   // sequencer 1
   INITIAL_STEP "No mode active":   // S1, max time T#10S, warning time T#7S
              N    #mode.activeMode:="mode_0_not_selected"
   END_STEP
   TRANSITION Trans1 FROM "No mode active" TO "Return to base position active"   // T1
      := #mode.button.basic.request.visibility AND #mode.button.basic.request.button;
   END_TRANSITION
   TRANSITION Trans6 FROM "No mode active" TO "Manual mode active"   // T6
      := NOT #mode.switch.auto AND "DB_Eks_Instance".Status.Global.AnyValidKey AND #iSafetyOKmanual;
   END_TRANSITION
   STEP "Return to base position active":   // S2, max time T#10S, warning time T#7S
              N    #mode.activeMode:="mode_2_base"
   END_STEP
   TRANSITION Trans2 FROM "Return to base position active" TO "Base position reached"   // T2
      := #iBasePosition;
   END_TRANSITION
   TRANSITION Trans5 FROM "Return to base position active" TO Done   // T5
      := NOT #iSafetyOKauto OR ((NOT #iBaseInManualMode OR #mode.switch.poloautomaActivated) AND NOT #mode.switch.auto) OR (#iBaseInManualMode AND #mode.switch.auto AND NOT #mode.switch.poloautomaActivated) OR #F_TRIG_semiauto_switch.Q;
   END_TRANSITION
   STEP "Base position reached":   // S3, max time T#10S, warning time T#7S
              N    #mode.activeMode:="mode_2_base"
   END_STEP
   TRANSITION Trans3 FROM "Base position reached" TO "Automatic mode active"   // T3
      := (#mode.button.auto.startRequest.visibility AND #mode.button.auto.startRequest.button) OR #mode.switch.poloautomaActivated;
   END_TRANSITION
   TRANSITION Trans8 FROM "Base position reached" TO Done   // T8
      := NOT #iSafetyOKauto OR (NOT #iBaseInManualMode AND NOT #mode.switch.auto) OR NOT #iBasePosition OR #F_TRIG_switchAuto.Q;
   END_TRANSITION
   STEP "Automatic mode active":   // S4, max time T#10S, warning time T#7S
              N    #mode.activeMode:="mode_3_automat"
   END_STEP
   TRANSITION Trans4 FROM "Automatic mode active" TO Done   // T4
      := NOT "AlwaysTRUE";
   END_TRANSITION
   TRANSITION Trans9 FROM "Automatic mode active" TO Done   // T9
      := NOT #iSafetyOKauto OR NOT #mode.switch.auto;
   END_TRANSITION
   TRANSITION Trans12 FROM "Automatic mode active" TO "R1 EXT off during auto"   // T12
      := NOT "iR1ext";
   END_TRANSITION
   STEP "Manual mode active":   // S5, max time T#10S, warning time T#7S
              N    #mode.activeMode:="mode_1_manual"
   END_STEP
   TRANSITION Trans7 FROM "Manual mode active" TO Done   // T7
      := #mode.switch.auto OR NOT "DB_Eks_Instance".Status.Global.AnyValidKey OR NOT #iSafetyOKmanual;
   END_TRANSITION
   TRANSITION Trans10 FROM "Manual mode active" TO "Return to base position active"   // T10, jump
      := #mode.button.basic.request.visibility AND #mode.button.basic.request.button;
   END_TRANSITION
   STEP Done:   // S6, max time T#10S, warning time T#7S
   END_STEP
   TRANSITION Trans11 FROM Done TO "No mode active"   // T11, jump
      := TRUE;
   END_TRANSITION
   STEP "R1 EXT off during auto":   // S7, max time T#10S, warning time T#7S
   END_STEP
   TRANSITION Trans13 FROM "R1 EXT off during auto" TO Done   // T13
      := TRUE;
   END_TRANSITION

   // permanent post-instructions
   NETWORK 1
   TITLE = semiauto mode
      IF ((#mode.activeMode = "mode_2_base") OR (#mode.activeMode = "mode_3_automat")) AND #mode.switch.poloautomaActivated THEN
          #mode.activeMode := "mode_4_semiautomat";
      END_IF;
   NETWORK 2
   TITLE = previous mode
      #mode.modeChanged := #mode.activeMode <> #PrevMode;
      #PrevMode := #mode.activeMode;
END_FUNCTION_BLOCK

FUNCTION_BLOCK "Lamps"   // FB7, LAD
{ S7_Optimized_Access := 'TRUE' }
VERSION : 0.1
// stored: AutoNumber true, IsIECCheckEnabled false, IsRetainMemResEnabled false, MemoryReserve 100, SetENOAutomatically false, UDAEnableTagReadback false
   VAR
      R_TRIG_Instance { S7_SetPoint := 'True'} : R_TRIG;
      IEC_Timer_0_Instance { S7_SetPoint := 'True'} : TON_TIME;
   END_VAR
BEGIN

REGION Network 1: Lighthouse lamps
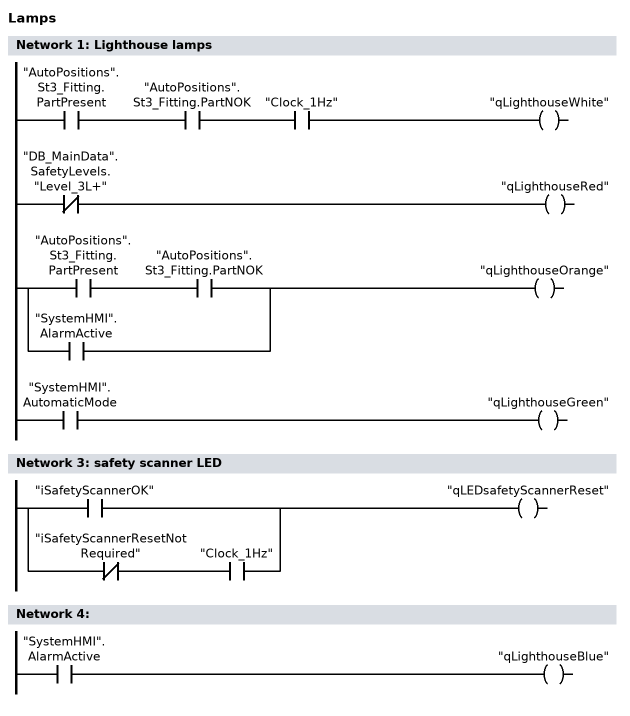
   RUNG wire#powerrail
      Contact( "AutoPositions".St3_Fitting.PartPresent )
      Contact( "AutoPositions".St3_Fitting.PartNOK )
      Contact( "Clock_1Hz" )
      Coil( "qLighthouseWhite" )
   END_RUNG
   RUNG wire#powerrail
      I_Contact( "DB_MainData".SafetyLevels."Level_3L+" )
      Coil( "qLighthouseRed" )
   END_RUNG
   RUNG wire#powerrail
      Contact( "AutoPositions".St3_Fitting.PartPresent )
      Contact( "AutoPositions".St3_Fitting.PartNOK )
      wire#w1
      Coil( "qLighthouseOrange" )
   END_RUNG
   RUNG wire#powerrail
      Contact( "SystemHMI".AlarmActive )
   END_RUNG wire#w1
   RUNG wire#powerrail
      Contact( "SystemHMI".AutomaticMode )
      Coil( "qLighthouseGreen" )
   END_RUNG
   // the same network as SCL:
   "qLighthouseWhite" := "AutoPositions".St3_Fitting.PartPresent AND "AutoPositions".St3_Fitting.PartNOK AND "Clock_1Hz";
   "qLighthouseRed" := NOT "DB_MainData".SafetyLevels."Level_3L+";
   "qLighthouseOrange" := ("AutoPositions".St3_Fitting.PartPresent AND "AutoPositions".St3_Fitting.PartNOK) OR "SystemHMI".AlarmActive;
   "qLighthouseGreen" := "SystemHMI".AutomaticMode;
END_REGION

REGION Network 2 (SCL): Alarm LED on OP
   //red button hmi
   "qResetAlarm" := "SystemHMI".AlarmActiveBlinking  AND "Clock_1Hz";
END_REGION

REGION Network 3: safety scanner LED
   RUNG wire#powerrail
      Contact( "iSafetyScannerOK" )
      wire#w1
      Coil( "qLEDsafetyScannerReset" )
   END_RUNG
   RUNG wire#powerrail
      I_Contact( "iSafetyScannerResetNotRequired" )
      Contact( "Clock_1Hz" )
   END_RUNG wire#w1
   // the same network as SCL:
   "qLEDsafetyScannerReset" := "iSafetyScannerOK" OR (NOT "iSafetyScannerResetNotRequired" AND "Clock_1Hz");
END_REGION

REGION Network 4
   RUNG wire#powerrail
      Contact( "SystemHMI".AlarmActive )
      Coil( "qLighthouseBlue" )
   END_RUNG
   // the same network as SCL:
   "qLighthouseBlue" := "SystemHMI".AlarmActive;
END_REGION
END_FUNCTION_BLOCK

FUNCTION "FC_READING_MAIN" : Void   // FC304, LAD
{ S7_Optimized_Access := 'TRUE' }
VERSION : 0.1
// stored: AutoNumber false, IsIECCheckEnabled false, SetENOAutomatically false, UDAEnableTagReadback false
BEGIN

REGION Network 1: Dataman readers block calls
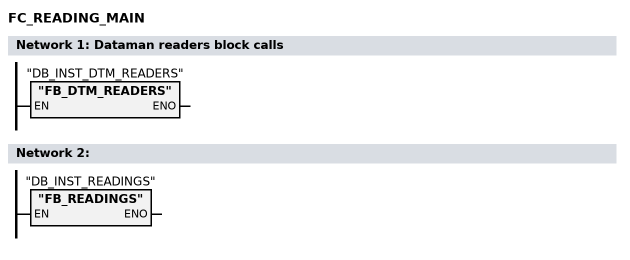
   RUNG wire#powerrail
      "DB_INST_DTM_READERS"()
   END_RUNG
   // the same network as SCL:
   "DB_INST_DTM_READERS"();   // "FB_DTM_READERS"
END_REGION

REGION Network 2
   RUNG wire#powerrail
      "DB_INST_READINGS"()
   END_RUNG
   // the same network as SCL:
   "DB_INST_READINGS"();   // "FB_READINGS"
END_REGION
END_FUNCTION

FUNCTION_BLOCK "FB_DTM_READERS"
{ S7_Optimized_Access := 'TRUE' }
VERSION : 0.1
   VAR 
      READER { S7_SetPoint := 'False'} : Array[1..5] of "FB_DTM";
   END_VAR


BEGIN
	//Call block reader 1
	#READER[1](TriggerReady:= "DM_SMLH-TriggerReady",
	           TriggerAck:="DM_SMLH-TriggerAck",
	           ResultsAvailable:="DM_SMLH-Results Available",
	           ResultID:="DM_SMLH-ResultID",
	           ResultCode:="DM_SMLH-Result Code",
	           ResultLenght:="DM_SMLH-Result Length",
	           ResultData:="DM_SMLH-ResultData",
	           TriggerEnable=>"DM_SMLH-TriggerEnable",
	           Trigger=>"DM_SMLH-Trigger",
	           ResultsAck=>"DM_SMLH-ResultsAck"
	          );
	
	//Call block reader 2
	          #READER[2](TriggerReady := "DM_SMRH-TriggerReady",
	           TriggerAck := "DM_SMRH-TriggerAck",
	           ResultsAvailable := "DM_SMRH-Results Available",
	           ResultID := "DM_SMRH-ResultID",
	           ResultCode := "DM_SMRH-Result Code",
	           ResultLenght := "DM_SMRH-Result Length",
	           ResultData := "DM_SMRH-ResultData",
	           TriggerEnable => "DM_SMRH-TriggerEnable",
	           Trigger => "DM_SMRH-Trigger",
	           ResultsAck => "DM_SMRH-ResultsAck"
	           );
	
	//Call block reader 3
	           #READER[3](TriggerReady:= "DM_FT-TriggerReady",
	           TriggerAck := "DM_FT-TriggerAck",
	           ResultsAvailable := "DM_FT-Results Available",
	           ResultID := "DM_FT-ResultID",
	           ResultCode := "DM_FT-Result Code",
	           ResultLenght := "DM_FT-Result Length",
	           ResultData := "DM_FT-ResultData",
	           TriggerEnable => "DM_FT-TriggerEnable",
	           Trigger => "DM_FT-Trigger",
	           ResultsAck => "DM_FT-ResultsAck");
	
	//Call block reader 4
	#READER[4](TriggerReady:= "DM_RT-TriggerReady",
	           TriggerAck := "DM_RT-TriggerAck",
	           ResultsAvailable := "DM_RT-Results Available",
	           ResultID := "DM_RT-ResultID",
	           ResultCode := "DM_RT-Result Code",
	           ResultLenght := "DM_RT-Result Length",
	           ResultData := "DM_RT-ResultData",
	           TriggerEnable => "DM_RT-TriggerEnable",
	           Trigger => "DM_RT-Trigger",
	           ResultsAck => "DM_RT-ResultsAck");
	
	
END_FUNCTION_BLOCK

FUNCTION_BLOCK "FB_DTM"   // FB301, LAD
{ S7_Optimized_Access := 'TRUE' }
VERSION : 0.1
// stored: AutoNumber false, IsIECCheckEnabled false, IsRetainMemResEnabled false, MemoryReserve 100, SetENOAutomatically false, UDAEnableTagReadback false
   VAR_INPUT
      Req : Bool;
      TriggerReady : Bool;
      TriggerAck : Bool;
      ResultsAvailable : Bool;
      ResultID : Word;
      ResultCode : Word;
      ResultLenght : Word;
      ResultData : "udt_DTM_resultData";
   END_VAR
   VAR_OUTPUT
      TriggerEnable : Bool;
      Trigger : Bool;
      ResultsAck : Bool;
      DataStr : String;
   END_VAR
   VAR
      ResultPending { ExternalAccessible := 'False'; ExternalVisible := 'False'; ExternalWritable := 'False'} : Bool;
      LatestResults { ExternalAccessible := 'False'; ExternalVisible := 'False'; ExternalWritable := 'False'} : Struct
         ID { ExternalAccessible := 'False'; ExternalVisible := 'False'; ExternalWritable := 'False'} : Int;
         Flags { ExternalAccessible := 'False'; ExternalVisible := 'False'; ExternalWritable := 'False'} : Int;
         Length { ExternalAccessible := 'False'; ExternalVisible := 'False'; ExternalWritable := 'False'} : Int;
         Value { ExternalAccessible := 'False'; ExternalVisible := 'False'; ExternalWritable := 'False'} : Array[0..63] of Byte;
      END_STRUCT;
   END_VAR
   VAR CONSTANT
      test : Bool := true;
   END_VAR
   VAR_TEMP   // added for the SCL form of the ladder/FBD networks
      _w1 : Bool;
   END_VAR
BEGIN

REGION Network 1: DataMan Acquisition Control Module
   // Make sure triggering is enabled
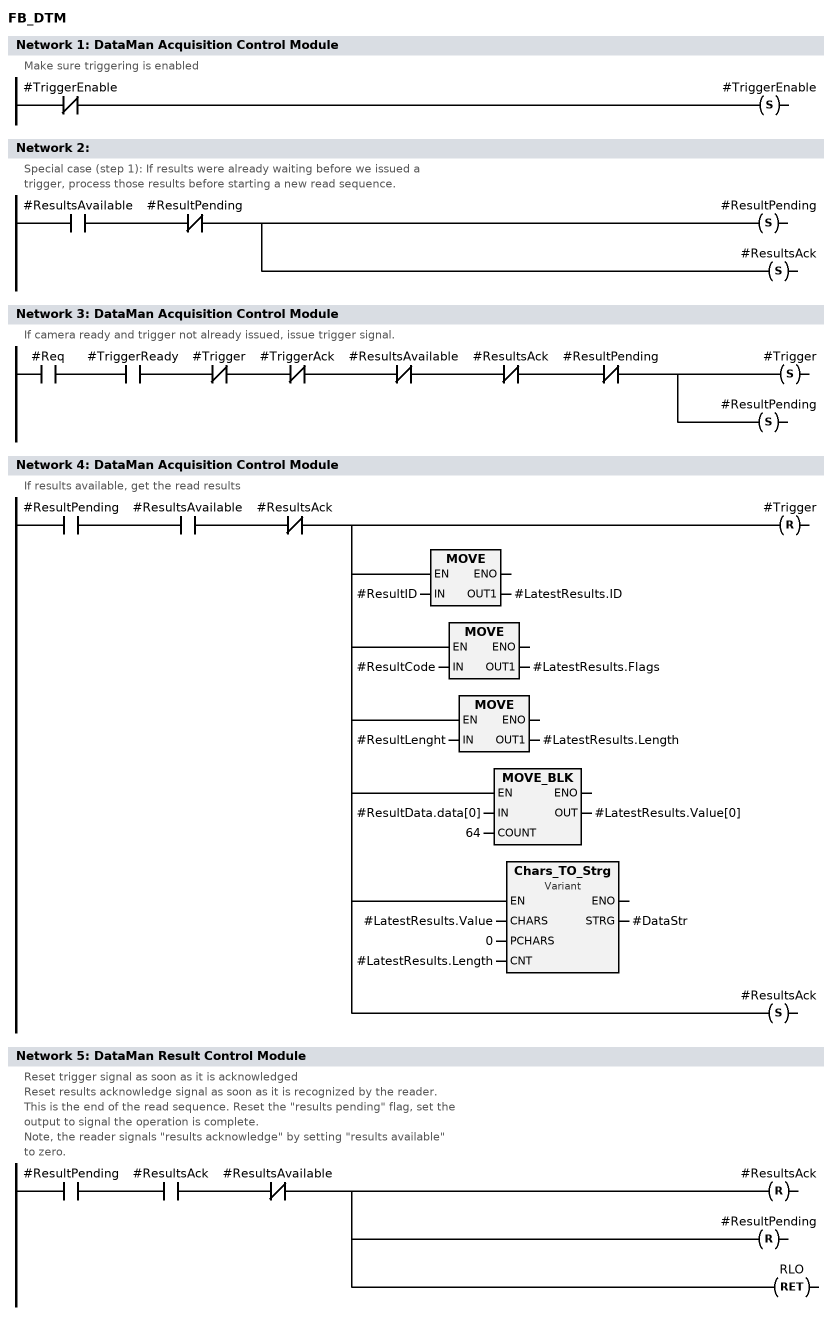
   RUNG wire#powerrail
      I_Contact( #TriggerEnable )
      S_Coil( #TriggerEnable )
   END_RUNG
   // the same network as SCL:
   IF NOT #TriggerEnable THEN #TriggerEnable := TRUE; END_IF;
END_REGION

REGION Network 2
   // Special case (step 1): If results were already waiting before we issued a 
   // trigger, process those results before starting a new read sequence.
   RUNG wire#powerrail
      Contact( #ResultsAvailable )
      I_Contact( #ResultPending )
      wire#w1
      S_Coil( #ResultPending )
   END_RUNG
   RUNG wire#w1
      S_Coil( #ResultsAck )
   END_RUNG
   // the same network as SCL:
   #_w1 := #ResultsAvailable AND NOT #ResultPending;
   IF #_w1 THEN
       #ResultPending := TRUE;
       #ResultsAck := TRUE;
   END_IF;
END_REGION

REGION Network 3: DataMan Acquisition Control Module
   // If camera ready and trigger not already issued, issue trigger signal.
   RUNG wire#powerrail
      Contact( #Req )
      Contact( #TriggerReady )
      I_Contact( #Trigger )
      I_Contact( #TriggerAck )
      I_Contact( #ResultsAvailable )
      I_Contact( #ResultsAck )
      I_Contact( #ResultPending )
      wire#w1
      S_Coil( #Trigger )
   END_RUNG
   RUNG wire#w1
      S_Coil( #ResultPending )
   END_RUNG
   // the same network as SCL:
   #_w1 := #Req AND #TriggerReady AND NOT #Trigger AND NOT #TriggerAck AND NOT #ResultsAvailable AND NOT #ResultsAck AND NOT #ResultPending;
   IF #_w1 THEN
       #Trigger := TRUE;
       #ResultPending := TRUE;
   END_IF;
END_REGION

REGION Network 4: DataMan Acquisition Control Module
   // If results available, get the read results
   IF #ResultPending AND #ResultsAvailable AND NOT #ResultsAck THEN
       #Trigger := FALSE;
       #LatestResults.ID := #ResultID;
       #LatestResults.Flags := #ResultCode;
       #LatestResults.Length := #ResultLenght;
       MOVE_BLK(IN := #ResultData.data[0], COUNT := 64, OUT => #LatestResults.Value[0]);
       Chars_TO_Strg(Chars := #LatestResults.Value, pChars := 0, Cnt := #LatestResults.Length, Strg => #DataStr);
       #ResultsAck := TRUE;
   END_IF;
END_REGION

REGION Network 5: DataMan Result Control Module
   // Reset trigger signal as soon as it is acknowledged 
   // Reset results acknowledge signal as soon as it is recognized by the reader.
   // 
   // This is the end of the read sequence. Reset the "results pending" flag, set the 
   // output to signal the operation is complete.
   // 
   // Note, the reader signals "results acknowledge" by setting "results available" 
   // to zero.
   #_w1 := #ResultPending AND #ResultsAck AND NOT #ResultsAvailable;
   IF #_w1 THEN
       #ResultsAck := FALSE;
       #ResultPending := FALSE;
       ENO := TRUE;
       RETURN;
   END_IF;
END_REGION
END_FUNCTION_BLOCK

FUNCTION_BLOCK "FB_READINGS"
{ S7_Optimized_Access := 'FALSE' }
VERSION : 0.1
   VAR 
      Reading : Array[1.."MaxDataReading"] of Struct
         Done : Bool;
         OK : Bool;
         NOK : Bool;
         Scan : String[70];
         NFP : String[30];
         IJC : Array[1.."NumberOfmessages"] of Struct
            SendMsg : Bool;
            Done : Bool;
            Answer : Int;
            State : USInt;
         END_STRUCT;
      END_STRUCT;
      ReadingsDone : Bool;
      Errors : Array[1..2] of Word;
      Error { ExternalAccessible := 'False'; ExternalVisible := 'False'; ExternalWritable := 'False'} AT Errors : Array[1..2, 1..16] of Bool;
   END_VAR

   VAR_TEMP 
      lctr1 : Int;
      lctr2 : Int;
      tempHolder : String;
      blankStr : String;
      NumberOfReadings : Int;
      eType : Int;   // Error type 1:reading, 2:IJCore
      count : Int;
   END_VAR

   VAR CONSTANT 
      NotUsed : USInt := 0;
      MasterNFP : USInt := 2;
      SecondaryNFP : USInt := 3;
      Component : USInt := 4;
   END_VAR


BEGIN
	//TITLE = 'READINGS'
	//AUTHOR: RAUL ROBINS
	//CREATED ON: 03/24/2023
	//VERSION: 1.0
	
	#NumberOfReadings := "DB_ProductionProgramActual".Program.NumberOfReadings;
	
	REGION Read code
	    
	    //Read request
	    IF "DevicesData".scanner.start THEN
	        FOR #lctr1 := 1 TO #NumberOfReadings DO
	            IF "DB_ProductionProgramActual".Program.Readings[#lctr1].Enable AND
	                NOT #Reading[#lctr1].Done THEN
	                "DB_INST_DTM_READERS".READER["DB_ProductionProgramActual".Program.Readings[#lctr1].ReaderNumber].Req := TRUE;
	            END_IF;
	            IF "DB_INST_DTM_READERS".READER["DB_ProductionProgramActual".Program.Readings[#lctr1].ReaderNumber].ResultsAvailable AND
	                "DB_INST_DTM_READERS".READER["DB_ProductionProgramActual".Program.Readings[#lctr1].ReaderNumber].ResultLenght <> 0 THEN
	                "DB_INST_DTM_READERS".READER["DB_ProductionProgramActual".Program.Readings[#lctr1].ReaderNumber].Req := FALSE;
	                #Reading[#lctr1].Done := TRUE;
	            END_IF;
	            
	            //Results
	            IF #Reading[#lctr1].Done THEN
	                //Compare strings
	                #tempHolder := MID(IN := "DB_INST_DTM_READERS".READER["DB_ProductionProgramActual".Program.Readings[#lctr1].ReaderNumber].DataStr,
	                                   L := LEN("DB_ProductionProgramActual".Program.Readings[#lctr1].ReferenceToFound),
	                                   P := "DB_ProductionProgramActual".Program.Readings[#lctr1].ReferenceStartPosition);
	                
	                IF #tempHolder = "DB_ProductionProgramActual".Program.Readings[#lctr1].ReferenceToFound THEN
	                    //Results OK
	                    #Reading[#lctr1].Scan := "DB_INST_DTM_READERS".READER["DB_ProductionProgramActual".Program.Readings[#lctr1].ReaderNumber].DataStr;
	                    #Reading[#lctr1].OK := TRUE;
	                    #Reading[#lctr1].NOK := FALSE;
	                    
	                    
	                    //Copy  NFP 
	                    //Master NFP
	                    IF "DB_ProductionProgramActual".Program.Readings[#lctr1].LabelType = 2 THEN
	                        #Reading[#lctr1].NFP := LEFT(IN := "DB_INST_DTM_READERS".READER["DB_ProductionProgramActual".Program.Readings[#lctr1].ReaderNumber].DataStr, L := 30);
	                        //Secondary NFP
	                    ELSIF "DB_ProductionProgramActual".Program.Readings[#lctr1].LabelType = 3 THEN
	                        //Linked to created NFP
	                        IF "DB_ProductionProgramActual".Program.Readings[1].MasterReadingNumber > 0 THEN
	                            ;
	                            //Linked to readed NFP
	                        ELSIF "DB_ProductionProgramActual".Program.Readings[1].LinkedMasterNumber > 0 THEN
	                            #Reading[#lctr1].NFP := #Reading["DB_ProductionProgramActual".Program.Readings[#lctr1].LinkedMasterNumber].NFP;
	                        END_IF;
	                        
	                    END_IF;
	                ELSE
	                    //Results NOK
	                    #Reading[#lctr1].OK := FALSE;
	                    #Reading[#lctr1].NOK := TRUE;
	                    #Reading[#lctr1].Scan := #blankStr;
	                END_IF;
	            END_IF;
	            //Count readings ok
	            IF #Reading[#lctr1].OK AND (#Reading[#lctr1].Scan <> #blankStr) OR NOT "DB_ProductionProgramActual".Program.Readings[#lctr1].Enable THEN
	                #count += 1;
	            END_IF;
	            IF #count = "DB_ProductionProgramActual".Program.NumberOfReadings THEN
	                #ReadingsDone := TRUE;
	            END_IF;
	            //Copy readings to buffer data
	            IF "sq_carousel_insertion_st1"."Set part present".X THEN
	                "AutoPositions".St1_Table1.Readings[#lctr1].Scan := #Reading[#lctr1].Scan;
	            END_IF;
	            
	            
	        END_FOR;
	    END_IF;
	    
	    
	    
	END_REGION
	
	REGION IJCore
	    FOR #lctr1 := 1 TO #NumberOfReadings DO
	        //TRACE
	        FOR #lctr2 := 1 TO 5 DO
	            CASE "DB_ProductionProgramActual".Program.Readings[#lctr1].Message[#lctr2].MessageType OF
	                "STA":
	                    "FC_READING_IJC_STA"(Req := #Reading[#lctr1].OK,
	                                         MessageNumber := "DB_ProductionProgramActual".Program.Readings[#lctr1].Message[#lctr2].MessageFlagNumber,
	                                         TraceabilityMode := "DB_MAIN_IJCORE".Mode,
	                                         NFP := #Reading[#lctr1].Scan,
	                                         ErrReset := "AlwaysTRUE",
	                                         MessageDone => #Reading[#lctr1].IJC[#lctr2].Done,
	                                         Answer := #Reading[#lctr1].IJC[#lctr2].Answer,
	                                         State := #Reading[#lctr1].IJC[#lctr2].State);
	                    
	                "PFC":
	                    "FC_TRACE_PFC"(Req := "DB_MAIN_IJCORE".CMD.PFC,
	                                   MessageNumber := "DB_ProductionProgramActual".Program.Readings[#lctr1].Message[#lctr2].MessageFlagNumber,
	                                   TraceabilityMode := "DB_MAIN_IJCORE".Mode,
	                                   NFP := "AutoPositions".St3_Fitting.Readings["DB_ProductionProgramActual".Program.Readings[#lctr1].MasterReadingNumber].Scan,
	                                   Kanban := "DB_ProductionProgramActual".Program.FaureciaNumber,
	                                   ErrReset := TRUE,
	                                   MessageDone => #Reading[#lctr1].IJC[#lctr2].Done,
	                                   Answer => #Reading[#lctr1].IJC[#lctr2].Answer,
	                                   State := #Reading[#lctr1].IJC[#lctr2].State);
	                    
	                "TRR":
	                    "FC_TRACE_TRR"(Req := "DB_MAIN_IJCORE".CMD.TRR,
	                                   MessageNumber := "DB_ProductionProgramActual".Program.Readings[#lctr1].Message[#lctr2].MessageFlagNumber,
	                                   TraceabilityMode := "DB_MAIN_IJCORE".Mode,
	                                   NFP := "AutoPositions".St3_Fitting.Readings["DB_ProductionProgramActual".Program.Readings[#lctr1].MasterReadingNumber].Scan,
	                                   ProcessStatus := 1,
	                                   NumberOfProcess := 1,
	                                   ErrReset := TRUE,
	                                   MessageDone => #Reading[#lctr1].IJC[#lctr2].Done,
	                                   Answer => #Reading[#lctr1].IJC[#lctr2].Answer,
	                                   State := #Reading[#lctr1].IJC[#lctr2].State);
	                    
	                "TRC":
	                    IF "DB_ProductionProgramActual".Program.Readings[#lctr1].MasterReadingNumber > 0 THEN
	                        "FC_READING_IJC_TRC"(Req := "DB_MAIN_IJCORE".CMD.TRC,
	                                             MessageNumber := "DB_ProductionProgramActual".Program.Readings[#lctr1].Message[#lctr2].MessageFlagNumber,
	                                             TraceabilityMode := "DB_MAIN_IJCORE".Mode,
	                                             NFP := #Reading["DB_ProductionProgramActual".Program.Readings[#lctr1].MasterReadingNumber].Scan,
	                                             Scan := #Reading[#lctr1].Scan,
	                                             ErrReset := TRUE,
	                                             MessageDone => #Reading[#lctr1].IJC[#lctr2].Done,
	                                             Answer := #Reading[#lctr1].IJC[#lctr2].Answer,
	                                             State := #Reading[#lctr1].IJC[#lctr2].State);
	                    END_IF;
	                ELSE:
	                    ;
	                    
	            END_CASE;
	            
	        END_FOR;
	    END_FOR;
	    
	END_REGION
	
	
	
	
	REGION Clear Data
	    IF NOT "DevicesData".scanner.start THEN
	        FOR #lctr1 := 1 TO "MaxDataReading" DO
	            "DB_INST_DTM_READERS".READER["DB_ProductionProgramActual".Program.Readings[#lctr1].ReaderNumber].Req := FALSE;
	            #Reading[#lctr1].Done := FALSE;
	            #Reading[#lctr1].OK := FALSE;
	            #Reading[#lctr1].NOK := FALSE;
	            #ReadingsDone := FALSE;
	            #Reading[#lctr1].Scan := #blankStr;
	        END_FOR;
	    END_IF;
	END_REGION
	
	// REGION Error Management
	//     #eType := 1;
	//     FOR #lctr1 := 1 TO #NumberOfReadings DO
	//         IF #Reading[#lctr1].NOK THEN
	//             #Error[#eType, 1] := TRUE;
	//         END_IF;
	
	//         //IJCore Errors
	//         FOR #lctr2 := 1 TO "NumberOfIJCoreMessages" DO
	//             #eType := 2;
	//             CASE #Reading[#lctr1].IJC[#lctr2].Answer OF
	//                 -2:  // NFP not founded
	//                     #Error[#eType, 1] := TRUE;
	//                 -3:  //Part number NOT inside BOM
	//                     #Error[#eType, 2] := TRUE;
	//                 -4: // PFC not ok
	//                     #Error[#eType, 3] := TRUE;
	//                 -5: //Component already used
	//                     #Error[#eType, 4] := TRUE;
	//                 -6: //Module already used
	//                     #Error[#eType, 5] := true;
	//                 -10: //Status NOK from previous operation
	//                     #Error[#eType, 6] := true;
	//             END_CASE;
	//         END_FOR;
	//     END_FOR;
	
	//     FOR #lctr1 := 1 TO 2 DO
	//         #Errors[#lctr1] := SWAP(#Errors[#lctr1]);
	//     END_FOR;
	// END_REGION
	
	
	
	
	
	
END_FUNCTION_BLOCK

FUNCTION "FC_TRACE_TRR" : Void
{ S7_Optimized_Access := 'TRUE' }
VERSION : 0.1
   VAR_INPUT 
      Req : Bool;   // Request message
      MessageNumber : DInt;   // Message number
      TraceabilityMode : Int;   // Tracability mode
      NFP : String;
      ProcessStatus : USInt;
      NumberOfProcess : USInt;
      ErrReset : Bool;
   END_VAR

   VAR_OUTPUT 
      MessageDone : Bool;
      Answer : Int;
   END_VAR

   VAR_IN_OUT 
      State : USInt;
   END_VAR

   VAR_TEMP 
      SEND_OFFSET : Struct
         SW : DInt;
         MSG : DInt;
      END_STRUCT;
      REC_OFFSET : Struct
         SW : DInt;
         MSG : DInt;
         ANS : DInt;
      END_STRUCT;
      IDB : Int;
      i : Int;
      j : Int;
      k : Int;
      CNT : Int;
      CNT_STR : String[2];
      MSG : DInt;
      ErrCode : Int;
   END_VAR

   VAR CONSTANT 
      "DB" : Byte := 16#84;
      CLEAR : Word := 16#0000;
      MINUS1 : Word := 16#FFFF;
      PLUS1 : Word := 16#0001;
      DB_REC : DB_ANY := 1006;
      DB_SEND : DB_ANY := 1005;
      Blank : String := '';
   END_VAR


BEGIN
	//TITLE = 'IJCORE PROTOCOL'
	//AUTHOR: RAUL ROBINS
	//CREATED ON: 03/24/2023
	//VERSION: 3.0
	
	
	
	IF #MessageNumber < 1  THEN
	    RETURN;
	END_IF;
	
	
	
	
	IF NOT #Req THEN // Error Reset
	    #State := 0;
	END_IF;
	
	#SEND_OFFSET.SW := (#MessageNumber * 2) + 2; //Calc message send sw offset
	#SEND_OFFSET.MSG := ((#MessageNumber - 1) * 80) + 604; // Calc send message offset
	#REC_OFFSET.SW := (#MessageNumber - 1) * 2; // Calc receive sw offset
	#REC_OFFSET.ANS := ((#MessageNumber - 1) * 32) + 600; // Calc receive answer offset
	#REC_OFFSET.MSG := ((#MessageNumber - 1) * 32) + 602; // Calc receive message offset
	
	
	CASE #State OF
	    0: // Initial State
	        #MessageDone := FALSE;
	        #Answer := 0;
	
	        POKE(area := #DB, //Clear send flag
	             dbNumber := #DB_SEND,
	             byteOffset := #SEND_OFFSET.SW,
	             value := #MINUS1);
	        POKE(area := #DB, //Clear receive flag
	             dbNumber := #DB_REC,
	             byteOffset := #REC_OFFSET.SW,
	             value := #MINUS1);
	     
	        #State := 10; ///Transition to state 10
	        
	    10: // Wait for start command
	        IF #Req THEN //If start command active
	            
	            POKE(area := #DB, //Clear send flag
	                 dbNumber := #DB_SEND,
	                 byteOffset := #SEND_OFFSET.SW,
	                 value := #MINUS1);
	            POKE(area := #DB, //Clear receive flag
	                 dbNumber := #DB_REC,
	                 byteOffset := #REC_OFFSET.SW,
	                 value := #MINUS1);
	            POKE(area := #DB, // Clear answer 
	                 dbNumber := #DB_REC,
	                 byteOffset := #REC_OFFSET.ANS,
	                 value := #CLEAR);
	            
	            FOR #i := 0 TO 79 BY 1 DO //Clear all send array
	                POKE(area := #DB,
	                     dbNumber := #DB_SEND,
	                     byteOffset := (#SEND_OFFSET.MSG + #i),
	                     value := '$00');
	            END_FOR;
	            FOR #i := 0 TO 29 BY 1 DO //Clear all receive array
	                POKE(area := #DB,
	                     dbNumber := #DB_REC,
	                     byteOffset := (#REC_OFFSET.MSG + #i),
	                     value := '$00');
	            END_FOR;
	            #State := 20; //Transition to state 20
	        END_IF;
	        
	    20: // Create message to send
	        FOR #i := 0 TO 7 BY 1 DO //Copy NFP to DB to send
	            POKE(area := #DB,
	                 dbNumber := #DB_SEND,
	                 byteOffset := (#SEND_OFFSET.MSG + #i),
	                 value := #NFP[#i + 1]);
	        END_FOR;
	                
	  
	                
	                POKE(area := #DB, //Set the process status of the message
	                     dbNumber := #DB_SEND,
	                     byteOffset := (#SEND_OFFSET.MSG + 8),
	                     value := USINT_TO_CHAR(#ProcessStatus + 48));
	                
	          
	        #State := 30; // Transition to state 30
	        
	    30: //Set flag to "1" to inform that PLC is ready to send (DB5 Ó 1005)
	        POKE(area := #DB,//Set flag to "1" to inform that PLC is ready to send
	             dbNumber := #DB_SEND,
	             byteOffset := #SEND_OFFSET.SW,
	             value := #PLUS1);
	        #State := 40; // Transition to state 40
	        
	        
	    40: //Wait to IJCORE response with "-1"
	        IF (PEEK_WORD(area := #DB, dbNumber := #DB_SEND, byteOffset := #SEND_OFFSET.SW) = #MINUS1)
	        THEN
	            #State := 50; // Transition to state 50
	        END_IF;
	        
	    50: //Check if IJCORE have answer from DB Receive
	        IF (PEEK_WORD(area := #DB, dbNumber := #DB_REC, byteOffset := #REC_OFFSET.SW) = #PLUS1)
	        THEN
	            #Answer := WORD_TO_INT(PEEK_WORD(area := #DB, dbNumber := #DB_REC, byteOffset := #REC_OFFSET.ANS)); //Copy answer from IJCORE
	
	            #State := 60; // Transition to state 100
	        END_IF;
	        
	    60: //Change Flag to "-1"
	        POKE(area := #DB, //Set "-1" to IJCORE
	             dbNumber := #DB_REC,
	             byteOffset := #REC_OFFSET.SW,
	             value := #MINUS1);
	        #State := 100; // Transition to state 100
	        
	        
	    100: //Sequence done
	        CASE #TraceabilityMode OF
	            1:// Full traceability
	                IF #Answer = 1 THEN
	                    #MessageDone := TRUE;
	                ELSE
	                    #MessageDone := FALSE;
	                END_IF;
	            2:// Traceability only
	                #MessageDone := TRUE;
	        END_CASE;
	        
	        IF NOT #Req THEN
	            #State := 0; // Transition to state 0
	        END_IF;
	END_CASE;
	
	
	
	
	
	
	
END_FUNCTION

ORGANIZATION_BLOCK "Startup"   // OB124, LAD, Startup
TITLE = "Complete Restart"
{ S7_Optimized_Access := 'TRUE' }
VERSION : 0.1
// stored: AutoNumber true, IsIECCheckEnabled false, SetENOAutomatically false
   VAR_INPUT
      LostRetentive : Bool;   // True if retentive data are lost
      LostRTC : Bool;   // True if date and time are lost
   END_VAR
BEGIN

REGION Network 1: Braketest or mastering requred
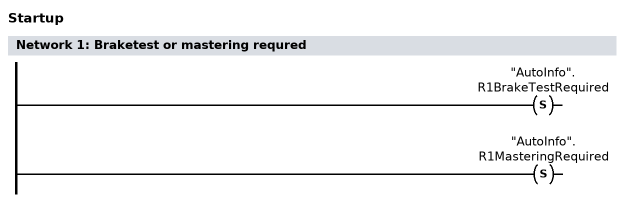
   RUNG wire#powerrail
      S_Coil( "AutoInfo".R1BrakeTestRequired )
   END_RUNG
   RUNG wire#powerrail
      S_Coil( "AutoInfo".R1MasteringRequired )
   END_RUNG
   // the same network as SCL:
   "AutoInfo".R1BrakeTestRequired := TRUE;
   "AutoInfo".R1MasteringRequired := TRUE;
END_REGION

REGION Network 2 (SCL)
       "DevicesData"."TA1-3MA".OverAcc := "StationParameters".Servo.OverAcc;
       "DevicesData"."TA1-3MA".OverDec := "StationParameters".Servo.OverDec;
       "DevicesData"."TA1-3MA".OverV := "StationParameters".Servo.OverV;
       "DevicesData"."TA1-3MA".Velocity := "StationParameters".Servo.Velocity;
END_REGION

REGION Network 3 (SCL)
   "setup_DB".minL := 100.0;
   "setup_DB".minR := "setup_DB".minL;
END_REGION
END_ORGANIZATION_BLOCK

ORGANIZATION_BLOCK "OB_IO_AccessError"   // OB122, LAD, IOAccessError
{ S7_Optimized_Access := 'TRUE' }
VERSION : 0.1
// stored: IsIECCheckEnabled false, SetENOAutomatically false
   VAR_INPUT
      BlockNr : UInt;   // Number of causing block
      Reaction : USInt;   // 0:ignore, 1:substitute, 2:skip
      Fault_ID : Byte;   // 16#42:reading, 16#43:writing
      BlockType : USInt;   // 16#01:OB, 16#02:FC, 16#03:FB, 16#04:SFC, 16#05:SFB, 16#06:DB: Type of block causing the error
      Area : USInt;   // 16#81:I, 16#82:Q: IO area where the IOaccess error occured
      DBNr : DB_ANY;   // Reserved for system
      Csg_OBNr : OB_ANY;   // Number of OB causing the error
      Csg_Prio : USInt;   // Priority of OB causing the error
      Width : USInt;   // 0:bit, 1:byte, 2:word, 3:dword, 4:lword
   END_VAR
BEGIN
END_ORGANIZATION_BLOCK

ORGANIZATION_BLOCK "OB_ProgrammingError"   // OB121, LAD, ProgrammingError
{ S7_Optimized_Access := 'TRUE' }
VERSION : 0.1
// stored: IsIECCheckEnabled false, SetENOAutomatically false
   VAR_INPUT
      BlockNr : UInt;   // Number of causing block
      Reaction : USInt;   // 0:ignore, 1:substitute, 2:skip
      Fault_ID : Byte;   // Fault identifier
      BlockType : USInt;   // 16#01:OB, 16#02:FC, 16#03:FB, 16#04:SFC, 16#05:SFB, 16#06:DB: Type of block causing the error
      Area : USInt;   // Area where the error occured
      DBNr : DB_ANY;   // DB number if Area = DB or DI
      Csg_OBNr : OB_ANY;   // Number of OB causing the error
      Csg_Prio : USInt;   // Priority of OB causing the error
      Width : USInt;   // 0:bit, 1:byte, 2:word, 3:dword, 4:lword
   END_VAR
BEGIN
END_ORGANIZATION_BLOCK

ORGANIZATION_BLOCK "OB_RackStationFailure"   // OB86, LAD, RackOrStationFailure
{ S7_Optimized_Access := 'TRUE' }
VERSION : 0.1
// stored: IsIECCheckEnabled false, SetENOAutomatically false
   VAR_INPUT
      LADDR : HW_DEVICE;   // Hardware identifier
      Event_Class : Byte;   // Event class
      Fault_ID : Byte;   // Fault identifier
   END_VAR
BEGIN
END_ORGANIZATION_BLOCK

ORGANIZATION_BLOCK "OB_Startup"   // OB100, LAD, Startup
TITLE = "Complete Restart"
{ S7_Optimized_Access := 'TRUE' }
VERSION : 0.1
// stored: AutoNumber true, IsIECCheckEnabled false, SetENOAutomatically false
   VAR_INPUT
      LostRetentive : Bool;   // True if retentive data are lost
      LostRTC : Bool;   // True if date and time are lost
   END_VAR
BEGIN
END_ORGANIZATION_BLOCK

ORGANIZATION_BLOCK "Diagnostic error interrupt"   // OB82, LAD, DiagnosticErrorInterrupt
{ S7_Optimized_Access := 'TRUE' }
VERSION : 0.1
// stored: IsIECCheckEnabled false, SetENOAutomatically false
   VAR_INPUT
      IO_State : Word;   // IO state of the HW object
      LADDR : HW_ANY;   // Hardware identifier
      Channel : UInt;   // Channel number
      MultiError : Bool;   // =true if more than one error is present
   END_VAR
BEGIN
END_ORGANIZATION_BLOCK

FUNCTION_BLOCK "CylinderINC"   // FB30, LAD
{ S7_Optimized_Access := 'FALSE' }
AUTHOR : Bodorik
FAMILY : RIV
NAME : Cylinder
VERSION : 0.9
// stored: AutoNumber false, IsIECCheckEnabled false, SetENOAutomatically false, UDAEnableTagReadback false
   VAR_INPUT
      POWER_OK : Bool;
      MOVE_BASIC : Bool;
      MOVE_WORK : Bool;
      MOVE_FREE : Bool;
      BASIC_POSITION : Bool;
      WORK_POSITION : Bool;
      TRIGGER : Bool;
      RESET : Bool;
      DELAY_BASIC : Time := T#1S;
      DELAY_WORK : Time := T#1S;
      DELAY_FREE : Time := T#1S;
      ERROR_TIME : Time := T#1S;
      ValveDelay : Time;
   END_VAR
   VAR_OUTPUT
      VALVE_BASIC : Bool;
      VALVE_WORK : Bool;
      CylinderStatus : "CylinderStatus";
      ERROR_BASIC : Bool;
      ERROR_WORK : Bool;
   END_VAR
   VAR_IN_OUT
      CylinderOperation : "CylinderOperation";
   END_VAR
   VAR DB_SPECIFIC
      "4l+Started" : Bool;
      InitCommandBP : Bool;
      InitCommandWP : Bool;
      BasicWorkStartWP : Bool;
      BasicWorkStartBP : Bool;
      work_valve : Bool;
      basic_valve : Bool;
      free_valve : Bool;
      baspos_error { S7_SetPoint := 'True'} : TON_TIME;
      workpos_error { S7_SetPoint := 'True'} : TON_TIME;
      baspos_delay { S7_SetPoint := 'True'} : TON_TIME;
      workpos_delay { S7_SetPoint := 'True'} : TON_TIME;
      CylinderOperationOld { S7_SetPoint := 'True'} : "CylinderOperation";
      IEC_Timer_0_Instance { S7_SetPoint := 'True'} : TP_TIME;
   END_VAR
   VAR
      R_TRIG_Instance { S7_SetPoint := 'True'} : R_TRIG;
   END_VAR
   VAR DB_SPECIFIC
      IEC_Timer_0_Instance_1 { S7_SetPoint := 'True'} : TP_TIME;
      IEC_Timer_0_Instance_2 { S7_SetPoint := 'True'} : TP_TIME;
      IEC_Timer_0_Instance_3 { S7_SetPoint := 'True'} : TON_TIME;
      IEC_Timer_0_Instance_4 { S7_SetPoint := 'True'} : TON_TIME;
   END_VAR
   VAR_TEMP
      et : Bool;
   END_VAR
   VAR_TEMP   // added for the SCL form of the ladder/FBD networks
      _w1 : Bool;
   END_VAR
BEGIN

REGION Network 1 (SCL): check new cylinder command
   //check if basic position req movement changed
   IF #CylinderOperation.ToBp <> #CylinderOperationOld.ToBp THEN
       #CylinderOperation.ToFp := false;
       #CylinderOperation.ToWp := false;
   END_IF;
   //check if work position req movement changed
   IF #CylinderOperation.ToWp <> #CylinderOperationOld.ToWp THEN
       #CylinderOperation.ToFp := false;
       #CylinderOperation.ToBp := false;
   END_IF;
   //check if free position req movement changed
   IF #CylinderOperation.ToFp <> #CylinderOperationOld.ToFp THEN
       #CylinderOperation.ToBp := false;
       #CylinderOperation.ToWp := false;
   END_IF;
   //store actual cylinder status to old
   #CylinderOperationOld := #CylinderOperation;
END_REGION

REGION Network 2: Start movement to basic position
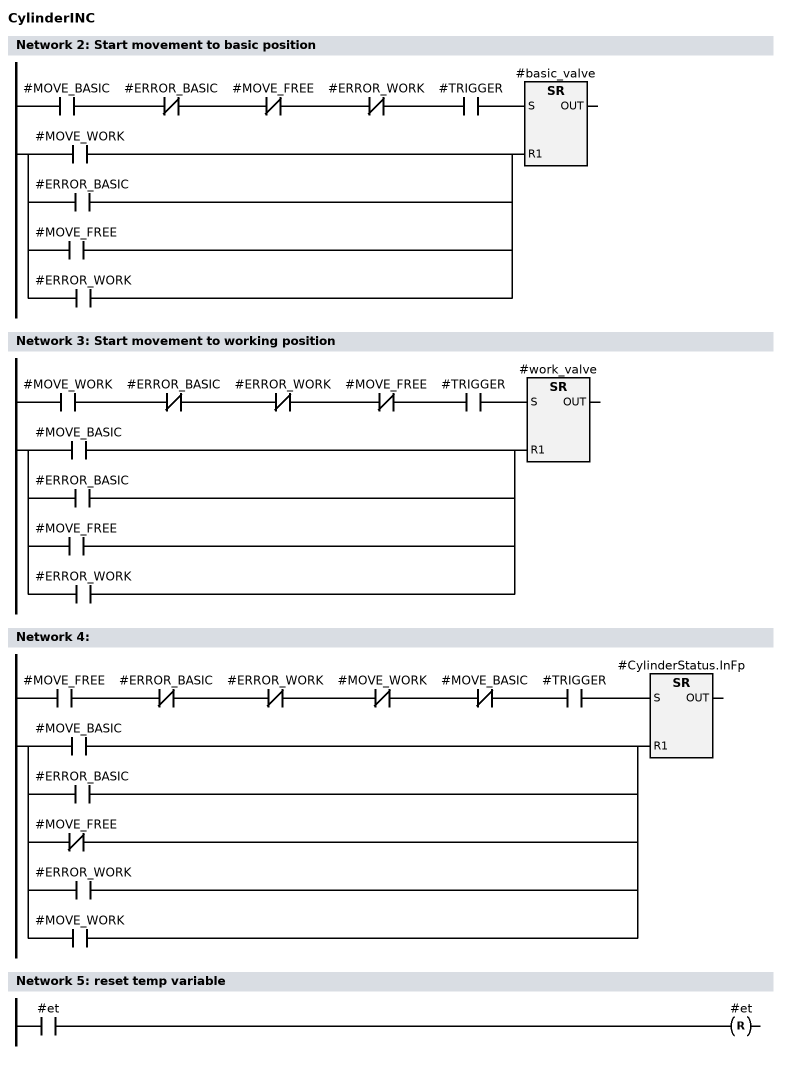
   RUNG wire#powerrail
      Contact( #MOVE_BASIC )
      I_Contact( #ERROR_BASIC )
      I_Contact( #MOVE_FREE )
      I_Contact( #ERROR_WORK )
      Contact( #TRIGGER )
      S_SR(operand := #basic_valve, r1 := wire#w1)
   END_RUNG
   RUNG wire#powerrail
      Contact( #MOVE_WORK )
   END_RUNG wire#w1
   RUNG wire#powerrail
      Contact( #ERROR_BASIC )
   END_RUNG wire#w1
   RUNG wire#powerrail
      Contact( #MOVE_FREE )
   END_RUNG wire#w1
   RUNG wire#powerrail
      Contact( #ERROR_WORK )
   END_RUNG wire#w1
   // the same network as SCL:
   IF #MOVE_BASIC AND NOT #ERROR_BASIC AND NOT #MOVE_FREE AND NOT #ERROR_WORK AND #TRIGGER THEN
       #basic_valve := TRUE;   // SR flip-flop
   END_IF;
   IF #MOVE_WORK OR #ERROR_BASIC OR #MOVE_FREE OR #ERROR_WORK THEN #basic_valve := FALSE; END_IF;
END_REGION

REGION Network 3: Start movement to working position
   RUNG wire#powerrail
      Contact( #MOVE_WORK )
      I_Contact( #ERROR_BASIC )
      I_Contact( #ERROR_WORK )
      I_Contact( #MOVE_FREE )
      Contact( #TRIGGER )
      S_SR(operand := #work_valve, r1 := wire#w1)
   END_RUNG
   RUNG wire#powerrail
      Contact( #MOVE_BASIC )
   END_RUNG wire#w1
   RUNG wire#powerrail
      Contact( #ERROR_BASIC )
   END_RUNG wire#w1
   RUNG wire#powerrail
      Contact( #MOVE_FREE )
   END_RUNG wire#w1
   RUNG wire#powerrail
      Contact( #ERROR_WORK )
   END_RUNG wire#w1
   // the same network as SCL:
   IF #MOVE_WORK AND NOT #ERROR_BASIC AND NOT #ERROR_WORK AND NOT #MOVE_FREE AND #TRIGGER THEN
       #work_valve := TRUE;   // SR flip-flop
   END_IF;
   IF #MOVE_BASIC OR #ERROR_BASIC OR #MOVE_FREE OR #ERROR_WORK THEN #work_valve := FALSE; END_IF;
END_REGION

REGION Network 4
   RUNG wire#powerrail
      Contact( #MOVE_FREE )
      I_Contact( #ERROR_BASIC )
      I_Contact( #ERROR_WORK )
      I_Contact( #MOVE_WORK )
      I_Contact( #MOVE_BASIC )
      Contact( #TRIGGER )
      S_SR(operand := #CylinderStatus.InFp, r1 := wire#w1)
   END_RUNG
   RUNG wire#powerrail
      Contact( #MOVE_BASIC )
   END_RUNG wire#w1
   RUNG wire#powerrail
      Contact( #ERROR_BASIC )
   END_RUNG wire#w1
   RUNG wire#powerrail
      I_Contact( #MOVE_FREE )
   END_RUNG wire#w1
   RUNG wire#powerrail
      Contact( #ERROR_WORK )
   END_RUNG wire#w1
   RUNG wire#powerrail
      Contact( #MOVE_WORK )
   END_RUNG wire#w1
   // the same network as SCL:
   IF #MOVE_FREE AND NOT #ERROR_BASIC AND NOT #ERROR_WORK AND NOT #MOVE_WORK AND NOT #MOVE_BASIC AND #TRIGGER THEN
       #CylinderStatus.InFp := TRUE;   // SR flip-flop
   END_IF;
   IF #MOVE_BASIC OR #ERROR_BASIC OR NOT #MOVE_FREE OR #ERROR_WORK OR #MOVE_WORK THEN
       #CylinderStatus.InFp := FALSE;
   END_IF;
END_REGION

REGION Network 5: reset temp variable
   RUNG wire#powerrail
      Contact( #et )
      R_Coil( #et )
   END_RUNG
   // the same network as SCL:
   IF #et THEN #et := FALSE; END_IF;
END_REGION

REGION Network 6 (FBD): Error movement to basic position
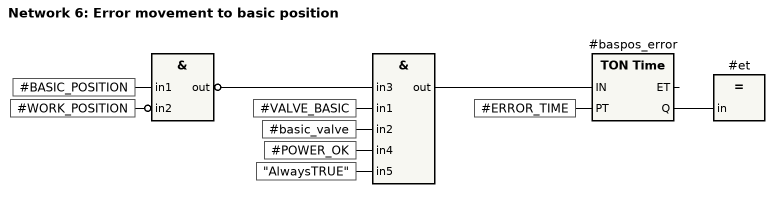
   #baspos_error(IN := NOT (#BASIC_POSITION AND NOT #WORK_POSITION) AND #VALVE_BASIC AND #basic_valve AND #POWER_OK AND "AlwaysTRUE",   // TON
                 PT := #ERROR_TIME);
   #et := #baspos_error.Q;
END_REGION

REGION Network 7: Set basic position error
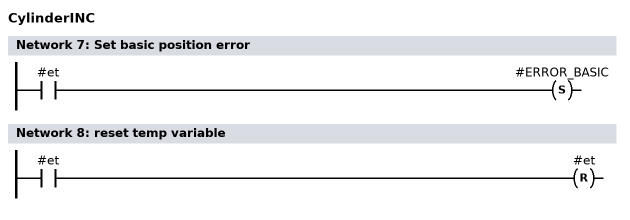
   RUNG wire#powerrail
      Contact( #et )
      S_Coil( #ERROR_BASIC )
   END_RUNG
   // the same network as SCL:
   IF #et THEN #ERROR_BASIC := TRUE; END_IF;
END_REGION

REGION Network 8: reset temp variable
   RUNG wire#powerrail
      Contact( #et )
      R_Coil( #et )
   END_RUNG
   // the same network as SCL:
   IF #et THEN #et := FALSE; END_IF;
END_REGION

REGION Network 9 (FBD): Error movement to working position
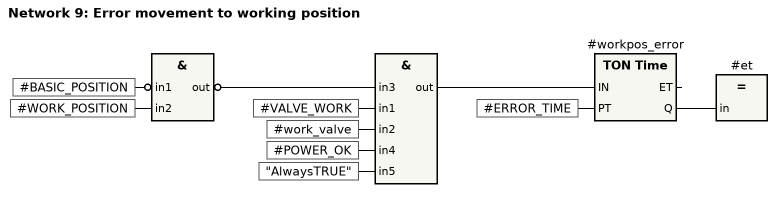
   #workpos_error(IN := NOT (NOT #BASIC_POSITION AND #WORK_POSITION) AND #VALVE_WORK AND #work_valve AND #POWER_OK AND "AlwaysTRUE",   // TON
                  PT := #ERROR_TIME);
   #et := #workpos_error.Q;
END_REGION

REGION Network 10: Set working position error
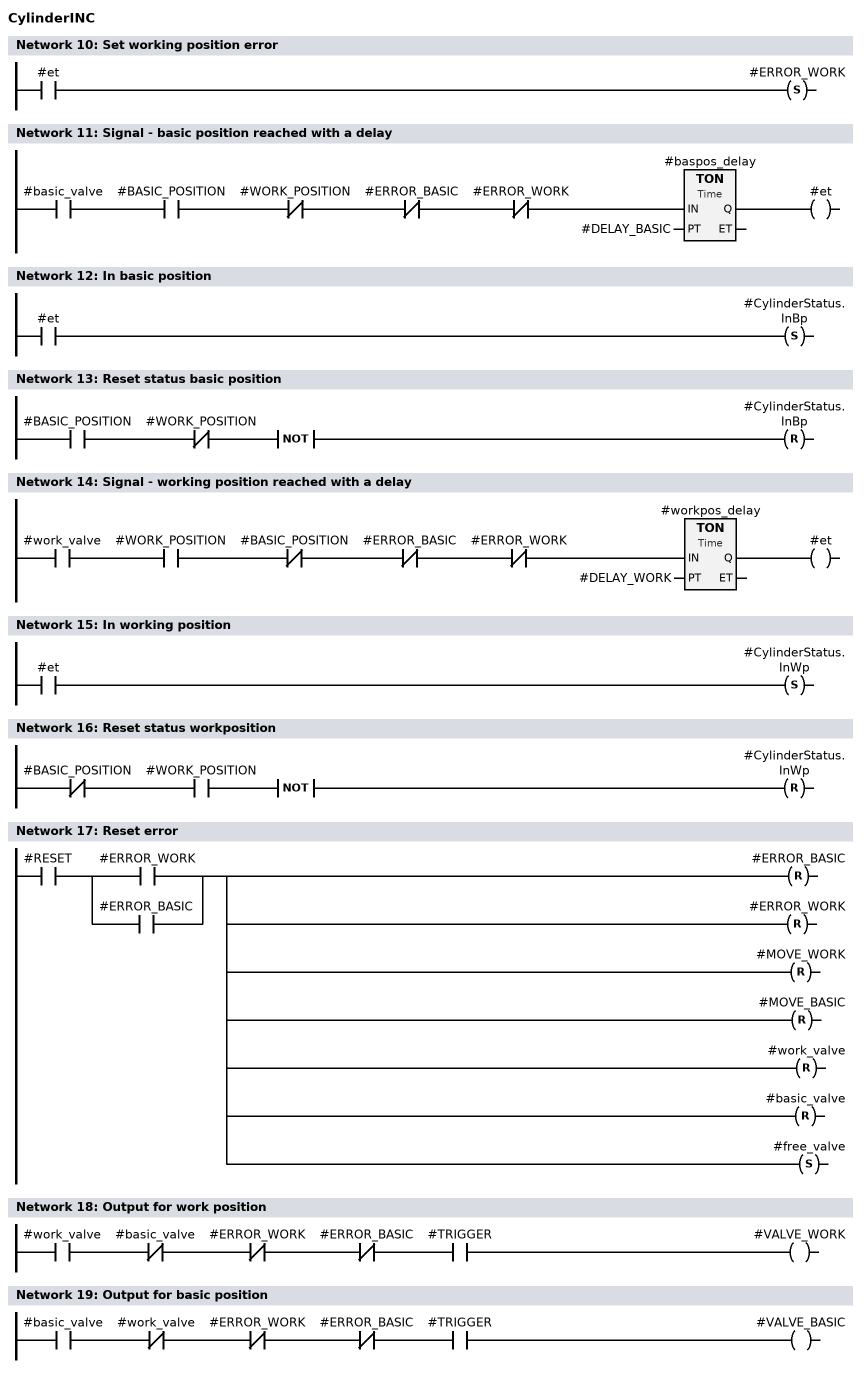
   RUNG wire#powerrail
      Contact( #et )
      S_Coil( #ERROR_WORK )
   END_RUNG
   // the same network as SCL:
   IF #et THEN #ERROR_WORK := TRUE; END_IF;
END_REGION

REGION Network 11: Signal - basic position reached with a delay
   RUNG wire#powerrail
      Contact( #basic_valve )
      Contact( #BASIC_POSITION )
      I_Contact( #WORK_POSITION )
      I_Contact( #ERROR_BASIC )
      I_Contact( #ERROR_WORK )
      { S7_Templates := "time_type := Time" } #baspos_delay.TON(pt := #DELAY_BASIC, et =>)
      Coil( #et )
   END_RUNG
   // the same network as SCL:
   #baspos_delay(PT := #DELAY_BASIC,   // TON
                 IN := #basic_valve AND #BASIC_POSITION AND NOT #WORK_POSITION AND NOT #ERROR_BASIC AND NOT #ERROR_WORK);
   #et := #baspos_delay.Q;
END_REGION

REGION Network 12: In basic position
   RUNG wire#powerrail
      Contact( #et )
      S_Coil( #CylinderStatus.InBp )
   END_RUNG
   // the same network as SCL:
   IF #et THEN #CylinderStatus.InBp := TRUE; END_IF;
END_REGION

REGION Network 13: Reset status basic position
   RUNG wire#powerrail
      Contact( #BASIC_POSITION )
      I_Contact( #WORK_POSITION )
      Not()
      R_Coil( #CylinderStatus.InBp )
   END_RUNG
   // the same network as SCL:
   IF NOT (#BASIC_POSITION AND NOT #WORK_POSITION) THEN #CylinderStatus.InBp := FALSE; END_IF;
END_REGION

REGION Network 14: Signal - working position reached with a delay
   RUNG wire#powerrail
      Contact( #work_valve )
      Contact( #WORK_POSITION )
      I_Contact( #BASIC_POSITION )
      I_Contact( #ERROR_BASIC )
      I_Contact( #ERROR_WORK )
      { S7_Templates := "time_type := Time" } #workpos_delay.TON(pt := #DELAY_WORK, et =>)
      Coil( #et )
   END_RUNG
   // the same network as SCL:
   #workpos_delay(PT := #DELAY_WORK,   // TON
                  IN := #work_valve AND #WORK_POSITION AND NOT #BASIC_POSITION AND NOT #ERROR_BASIC AND NOT #ERROR_WORK);
   #et := #workpos_delay.Q;
END_REGION

REGION Network 15: In working position
   RUNG wire#powerrail
      Contact( #et )
      S_Coil( #CylinderStatus.InWp )
   END_RUNG
   // the same network as SCL:
   IF #et THEN #CylinderStatus.InWp := TRUE; END_IF;
END_REGION

REGION Network 16: Reset status workposition
   RUNG wire#powerrail
      I_Contact( #BASIC_POSITION )
      Contact( #WORK_POSITION )
      Not()
      R_Coil( #CylinderStatus.InWp )
   END_RUNG
   // the same network as SCL:
   IF NOT (NOT #BASIC_POSITION AND #WORK_POSITION) THEN #CylinderStatus.InWp := FALSE; END_IF;
END_REGION

REGION Network 17: Reset error
   RUNG wire#powerrail
      Contact( #RESET )
      wire#w1
      Contact( #ERROR_WORK )
      wire#w2
      R_Coil( #ERROR_BASIC )
   END_RUNG
   RUNG wire#w1
      Contact( #ERROR_BASIC )
   END_RUNG wire#w2
   RUNG wire#w2
      R_Coil( #ERROR_WORK )
   END_RUNG
   RUNG wire#w2
      R_Coil( #MOVE_WORK )
   END_RUNG
   RUNG wire#w2
      R_Coil( #MOVE_BASIC )
   END_RUNG
   RUNG wire#w2
      R_Coil( #work_valve )
   END_RUNG
   RUNG wire#w2
      R_Coil( #basic_valve )
   END_RUNG
   RUNG wire#w2
      S_Coil( #free_valve )
   END_RUNG
   // the same network as SCL:
   #_w1 := #RESET AND (#ERROR_WORK OR #ERROR_BASIC);
   IF #_w1 THEN
       #ERROR_BASIC := FALSE;
       #ERROR_WORK := FALSE;
       #MOVE_WORK := FALSE;
       #MOVE_BASIC := FALSE;
       #work_valve := FALSE;
       #basic_valve := FALSE;
       #free_valve := TRUE;
   END_IF;
END_REGION

REGION Network 18: Output for work position
   RUNG wire#powerrail
      Contact( #work_valve )
      I_Contact( #basic_valve )
      I_Contact( #ERROR_WORK )
      I_Contact( #ERROR_BASIC )
      Contact( #TRIGGER )
      Coil( #VALVE_WORK )
   END_RUNG
   // the same network as SCL:
   #VALVE_WORK := #work_valve AND NOT #basic_valve AND NOT #ERROR_WORK AND NOT #ERROR_BASIC AND #TRIGGER;
END_REGION

REGION Network 19: Output for basic position
   RUNG wire#powerrail
      Contact( #basic_valve )
      I_Contact( #work_valve )
      I_Contact( #ERROR_WORK )
      I_Contact( #ERROR_BASIC )
      Contact( #TRIGGER )
      Coil( #VALVE_BASIC )
   END_RUNG
   // the same network as SCL:
   #VALVE_BASIC := #basic_valve AND NOT #work_valve AND NOT #ERROR_WORK AND NOT #ERROR_BASIC AND #TRIGGER;
END_REGION

REGION Network 20 (SCL)
   #R_TRIG_Instance(CLK:=#POWER_OK
   );

   IF #R_TRIG_Instance.Q THEN
       #"4l+Started" := TRUE;

   END_IF;

   IF #MOVE_BASIC AND #"4l+Started" THEN

       #InitCommandBP := true;
   END_IF;
   IF #MOVE_WORK AND #"4l+Started" THEN

       #InitCommandWP := true;
   END_IF;

   #IEC_Timer_0_Instance_1(IN:=#InitCommandBP,
                               PT:=t#10ms,
                               Q=>#BasicWorkStartBP
       );
   #IEC_Timer_0_Instance_2(IN:=#InitCommandWP,
                               PT:=t#10ms,
                               Q=>#BasicWorkStartWP
   );


   IF #BasicWorkStartBP  THEN
       #VALVE_WORK := TRUE;
       #VALVE_BASIC := FALSE;
       ;

   END_IF;

   IF #BasicWorkStartWP THEN
       #VALVE_WORK := FALSE;
       #VALVE_BASIC := TRUE;
       ;

   END_IF;

   IF NOT #IEC_Timer_0_Instance_1.Q AND #InitCommandBP THEN
       #VALVE_WORK := FALSE;
       #VALVE_BASIC := TRUE;
       #"4l+Started" := FALSE;
       #InitCommandBP := FALSE;
       ;
   END_IF;
   IF NOT #IEC_Timer_0_Instance_2.Q AND #InitCommandWP THEN
       #VALVE_WORK := TRUE;
       #VALVE_BASIC := FALSE;
       #"4l+Started" := FALSE;
       #InitCommandWP := FALSE;
       ;
   END_IF;
END_REGION
END_FUNCTION_BLOCK

FUNCTION "FC_ByteToCharacters" : Void   // FC1071, LAD
{ S7_Optimized_Access := 'FALSE' }
VERSION : 0.1
// stored: AutoNumber false, IsIECCheckEnabled false, SetENOAutomatically false, UDAEnableTagReadback false
   VAR_INPUT
      iByte : Byte;
   END_VAR
   VAR_OUTPUT
      qChar1 : Char;
      qChar2 : Char;
   END_VAR
   VAR_TEMP
      "b" : Byte;
      char1_value : UInt;
      char2_value : UInt;
   END_VAR
   VAR_TEMP   // added for the SCL form of the ladder/FBD networks
      _w1 : Bool;
      _w2 : Bool;
   END_VAR
BEGIN

REGION Network 1: Load input byte to temporary
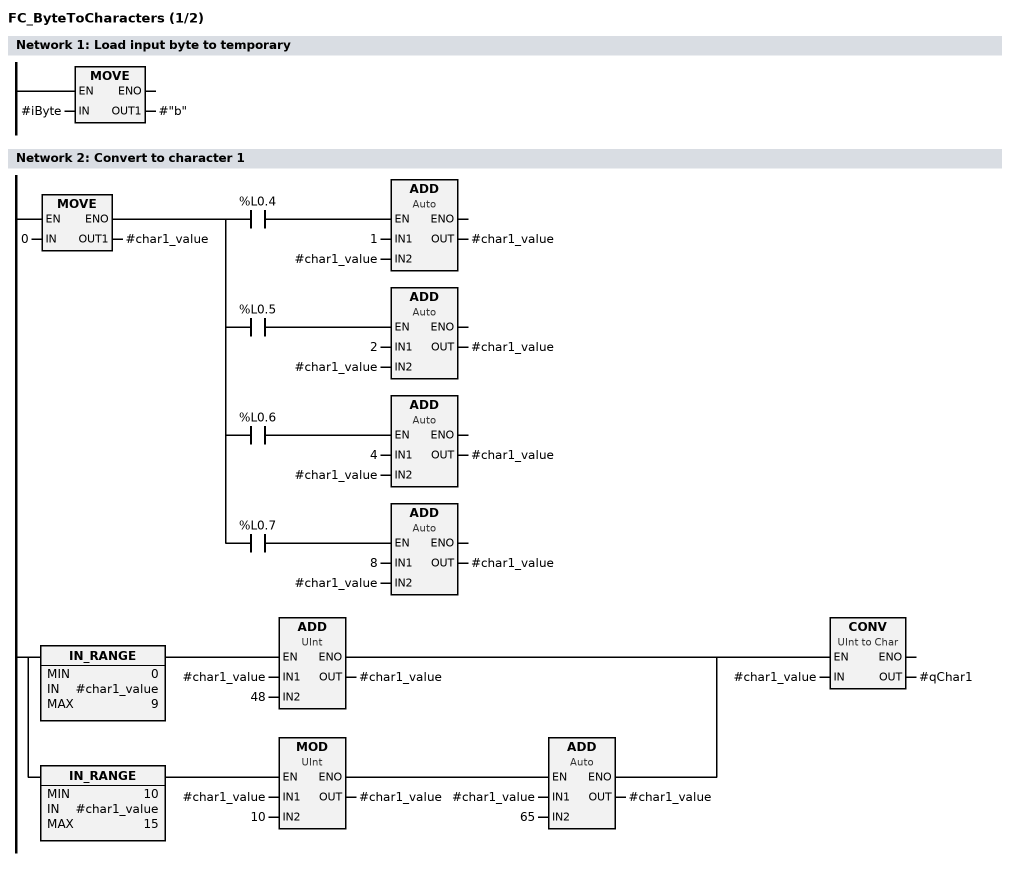
   RUNG wire#powerrail
      Move(in := #iByte, out1 => #"b")
   END_RUNG
   // the same network as SCL:
   #"b" := #iByte;
END_REGION

REGION Network 2: Convert to character 1
   RUNG wire#powerrail
      Move(in := 0, out1 => #char1_value)
      wire#w1
      Contact( %L0.4 )
      Add(in1 := 1, in2 := #char1_value, out => #char1_value)
   END_RUNG
   RUNG wire#w1
      Contact( %L0.5 )
      Add(in1 := 2, in2 := #char1_value, out => #char1_value)
   END_RUNG
   RUNG wire#w1
      Contact( %L0.6 )
      Add(in1 := 4, in2 := #char1_value, out => #char1_value)
   END_RUNG
   RUNG wire#w1
      Contact( %L0.7 )
      Add(in1 := 8, in2 := #char1_value, out => #char1_value)
   END_RUNG
   RUNG wire#powerrail
      { S7_Templates := "SrcType := UInt" } InRange(min := 0, in := #char1_value, max := 9)
      { S7_Templates := "SrcType := UInt" } Add(in1 := #char1_value, in2 := 48, out => #char1_value)
      wire#w2
      { S7_Templates := "[SrcType := UInt, DestType := Char]" } Convert(in := #char1_value, out => #qChar1)
   END_RUNG
   RUNG wire#powerrail
      { S7_Templates := "SrcType := UInt" } InRange(min := 10, in := #char1_value, max := 15)
      { S7_Templates := "SrcType := UInt" } Mod(in1 := #char1_value, in2 := 10, out => #char1_value)
      Add(in1 := #char1_value, in2 := 65, out => #char1_value)
   END_RUNG wire#w2
   // the same network as SCL:
   #char1_value := 0;
   IF %L0.4 THEN #char1_value := 1 + #char1_value; END_IF;
   IF %L0.5 THEN #char1_value := 2 + #char1_value; END_IF;
   IF %L0.6 THEN #char1_value := 4 + #char1_value; END_IF;
   IF %L0.7 THEN #char1_value := 8 + #char1_value; END_IF;
   #_w1 := (0 <= #char1_value) AND (#char1_value <= 9);
   IF #_w1 THEN #char1_value := #char1_value + 48; END_IF;
   #_w2 := (10 <= #char1_value) AND (#char1_value <= 15);
   IF #_w2 THEN
       #char1_value := #char1_value MOD 10;
       #char1_value := #char1_value + 65;
   END_IF;
   IF #_w1 OR #_w2 THEN #qChar1 := UINT_TO_CHAR(#char1_value); END_IF;
END_REGION

REGION Network 3: Convert to character 2
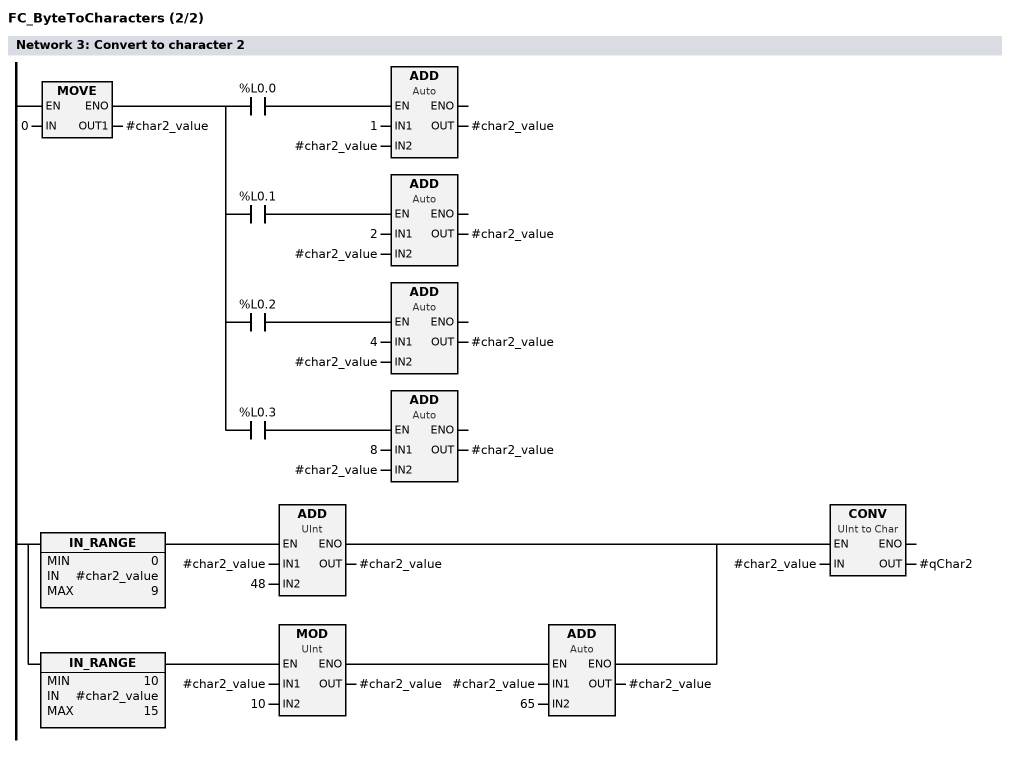
   RUNG wire#powerrail
      Move(in := 0, out1 => #char2_value)
      wire#w1
      Contact( %L0.0 )
      Add(in1 := 1, in2 := #char2_value, out => #char2_value)
   END_RUNG
   RUNG wire#w1
      Contact( %L0.1 )
      Add(in1 := 2, in2 := #char2_value, out => #char2_value)
   END_RUNG
   RUNG wire#w1
      Contact( %L0.2 )
      Add(in1 := 4, in2 := #char2_value, out => #char2_value)
   END_RUNG
   RUNG wire#w1
      Contact( %L0.3 )
      Add(in1 := 8, in2 := #char2_value, out => #char2_value)
   END_RUNG
   RUNG wire#powerrail
      { S7_Templates := "SrcType := UInt" } InRange(min := 0, in := #char2_value, max := 9)
      { S7_Templates := "SrcType := UInt" } Add(in1 := #char2_value, in2 := 48, out => #char2_value)
      wire#w2
      { S7_Templates := "[SrcType := UInt, DestType := Char]" } Convert(in := #char2_value, out => #qChar2)
   END_RUNG
   RUNG wire#powerrail
      { S7_Templates := "SrcType := UInt" } InRange(min := 10, in := #char2_value, max := 15)
      { S7_Templates := "SrcType := UInt" } Mod(in1 := #char2_value, in2 := 10, out => #char2_value)
      Add(in1 := #char2_value, in2 := 65, out => #char2_value)
   END_RUNG wire#w2
   // the same network as SCL:
   #char2_value := 0;
   IF %L0.0 THEN #char2_value := 1 + #char2_value; END_IF;
   IF %L0.1 THEN #char2_value := 2 + #char2_value; END_IF;
   IF %L0.2 THEN #char2_value := 4 + #char2_value; END_IF;
   IF %L0.3 THEN #char2_value := 8 + #char2_value; END_IF;
   #_w1 := (0 <= #char2_value) AND (#char2_value <= 9);
   IF #_w1 THEN #char2_value := #char2_value + 48; END_IF;
   #_w2 := (10 <= #char2_value) AND (#char2_value <= 15);
   IF #_w2 THEN
       #char2_value := #char2_value MOD 10;
       #char2_value := #char2_value + 65;
   END_IF;
   IF #_w1 OR #_w2 THEN #qChar2 := UINT_TO_CHAR(#char2_value); END_IF;
END_REGION
END_FUNCTION

FUNCTION_BLOCK "FB_IJC_AWAKE_SIGNAL"   // FB1003, LAD
TITLE = Awake signal
{ S7_Optimized_Access := 'TRUE' }
VERSION : 0.1
// This function supervise Awake signal, 
// - Awake signal is to test communication between PLC and IJCORE. 
// - Awake signal is set to 1 by PLC and set to -1 by IJCORE alternatively.
// - first PLC check if awake signal is different of 1, if it is, PLC launch timer T1 
//  (1s<T1<10s). at the end of this temporisation, PLC set awake signal to 1 and 
//  launch Timer 2. 
// - if IJCORE don't set awake signal to -1 before the end of timer 2,PLC generate  
//   Time out fault for awake signal.
// stored: AutoNumber false, IsIECCheckEnabled false, IsRetainMemResEnabled false, MemoryReserve 100, SetENOAutomatically false, UDAEnableTagReadback false
   VAR_INPUT
      ack_error : Bool;
   END_VAR
   VAR_OUTPUT
      State_com : SInt;
   END_VAR
   VAR
      T1PresetValue : Time := T#1S;
      T2PresetValue : Time := T#60S;
      AwSignalTimeOutFault : Bool := 0;
      Reset_Counters : Bool;
      Restart_Counter_bit_of_life : USInt := 0;
      NB_Bit_of_Life : Bool;
      number_restart : DInt;
      check_restart : Bool;
      "Timer" { ExternalAccessible := 'False'; ExternalVisible := 'False'; ExternalWritable := 'False'} : Array[1..5] of TON_TIME;
   END_VAR
   VAR CONSTANT
      Trestart : Time := T#200ms;
      T3 : Time := T#2s;
   END_VAR
   VAR_TEMP   // added for the SCL form of the ladder/FBD networks
      _w1 : Bool;
   END_VAR
BEGIN

REGION Network 1: - if awake signal is -1 then launch timer 1
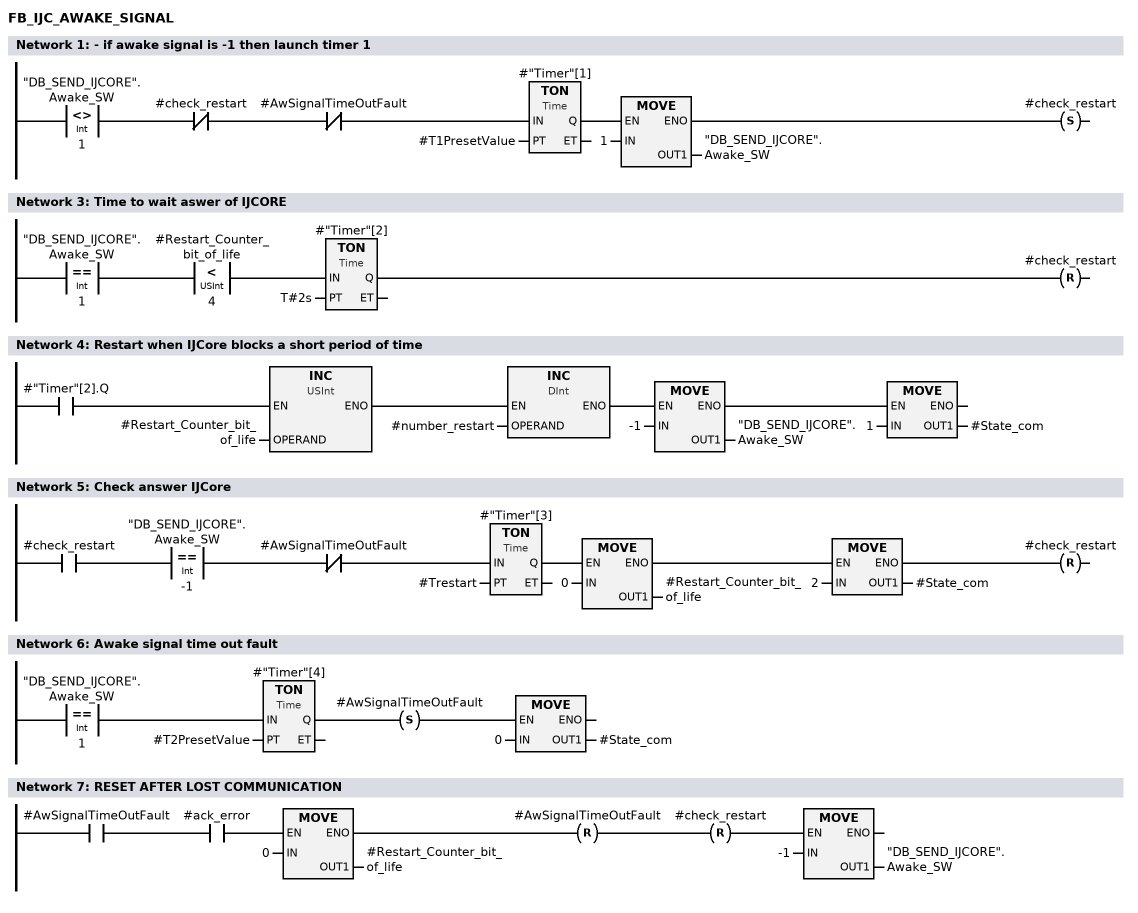
   RUNG wire#powerrail
      { S7_Templates := "SrcType := Int" } NE_Contact(in1 := "DB_SEND_IJCORE".Awake_SW, in2 := 1)
      I_Contact( #check_restart )
      I_Contact( #AwSignalTimeOutFault )
      { S7_Templates := "time_type := Time" } #"Timer"[1].TON(pt := #T1PresetValue, et =>)
      Move(in := 1, out1 => "DB_SEND_IJCORE".Awake_SW)
      S_Coil( #check_restart )
   END_RUNG
   // the same network as SCL:
   #"Timer"[1].TON(IN := ("DB_SEND_IJCORE".Awake_SW <> 1) AND NOT #check_restart AND NOT #AwSignalTimeOutFault,
                   PT := #T1PresetValue);
   IF #"Timer"[1].Q THEN
       "DB_SEND_IJCORE".Awake_SW := 1;
       #check_restart := TRUE;
   END_IF;
END_REGION

REGION Network 2: Diagnostic
END_REGION

REGION Network 3: Time to wait aswer of IJCORE
   RUNG wire#powerrail
      { S7_Templates := "SrcType := Int" } EQ_Contact(in1 := "DB_SEND_IJCORE".Awake_SW, in2 := 1)
      { S7_Templates := "SrcType := USInt" } LT_Contact(in1 := #Restart_Counter_bit_of_life, in2 := 4)
      { S7_Templates := "time_type := Time" } #"Timer"[2].TON(pt := T#2s, et =>)
      R_Coil( #check_restart )
   END_RUNG
   // the same network as SCL:
   #"Timer"[2].TON(IN := ("DB_SEND_IJCORE".Awake_SW = 1) AND (#Restart_Counter_bit_of_life < 4), PT := T#2s);
   IF #"Timer"[2].Q THEN #check_restart := FALSE; END_IF;
END_REGION

REGION Network 4: Restart when IJCore blocks a short period of time
   RUNG wire#powerrail
      Contact( #"Timer"[2].Q )
      { S7_Templates := "DestType := USInt" } Inc( #Restart_Counter_bit_of_life )
      { S7_Templates := "DestType := DInt" } Inc( #number_restart )
      Move(in := -1, out1 => "DB_SEND_IJCORE".Awake_SW)
      Move(in := 1, out1 => #State_com)
   END_RUNG
   // the same network as SCL:
   IF #"Timer"[2].Q THEN
       #Restart_Counter_bit_of_life := #Restart_Counter_bit_of_life + 1;
       #number_restart := #number_restart + 1;
       "DB_SEND_IJCORE".Awake_SW := -1;
       #State_com := 1;
   END_IF;
END_REGION

REGION Network 5: Check answer IJCore
   RUNG wire#powerrail
      Contact( #check_restart )
      { S7_Templates := "SrcType := Int" } EQ_Contact(in1 := "DB_SEND_IJCORE".Awake_SW, in2 := -1)
      I_Contact( #AwSignalTimeOutFault )
      { S7_Templates := "time_type := Time" } #"Timer"[3].TON(pt := #Trestart, et =>)
      Move(in := 0, out1 => #Restart_Counter_bit_of_life)
      Move(in := 2, out1 => #State_com)
      R_Coil( #check_restart )
   END_RUNG
   // the same network as SCL:
   #"Timer"[3].TON(IN := #check_restart AND ("DB_SEND_IJCORE".Awake_SW = (-1)) AND NOT #AwSignalTimeOutFault,
                   PT := #Trestart);
   IF #"Timer"[3].Q THEN
       #Restart_Counter_bit_of_life := 0;
       #State_com := 2;
       #check_restart := FALSE;
   END_IF;
END_REGION

REGION Network 6: Awake signal time out fault
   RUNG wire#powerrail
      { S7_Templates := "SrcType := Int" } EQ_Contact(in1 := "DB_SEND_IJCORE".Awake_SW, in2 := 1)
      { S7_Templates := "time_type := Time" } #"Timer"[4].TON(pt := #T2PresetValue, et =>)
      S_Coil( #AwSignalTimeOutFault )
      Move(in := 0, out1 => #State_com)
   END_RUNG
   // the same network as SCL:
   #"Timer"[4].TON(IN := "DB_SEND_IJCORE".Awake_SW = 1, PT := #T2PresetValue);
   IF #"Timer"[4].Q THEN
       #AwSignalTimeOutFault := TRUE;
       #State_com := 0;
   END_IF;
END_REGION

REGION Network 7: RESET AFTER LOST COMMUNICATION
   RUNG wire#powerrail
      Contact( #AwSignalTimeOutFault )
      Contact( #ack_error )
      Move(in := 0, out1 => #Restart_Counter_bit_of_life)
      R_Coil( #AwSignalTimeOutFault )
      R_Coil( #check_restart )
      Move(in := -1, out1 => "DB_SEND_IJCORE".Awake_SW)
   END_RUNG
   // the same network as SCL:
   IF #AwSignalTimeOutFault AND #ack_error THEN #Restart_Counter_bit_of_life := 0; END_IF;
   #_w1 := #AwSignalTimeOutFault AND #ack_error;
   IF #_w1 THEN
       #AwSignalTimeOutFault := FALSE;
       #check_restart := FALSE;
       "DB_SEND_IJCORE".Awake_SW := -1;
   END_IF;
END_REGION
END_FUNCTION_BLOCK

FUNCTION_BLOCK "Main_Safety_RTG1"   // FB0, F_LAD
{ S7_Optimized_Access := 'TRUE' }
VERSION : 0.1
// stored: AutoNumber false, IsIECCheckEnabled false, UDAEnableTagReadback false
   VAR
      ACK_GL_Instance : ACK_GL;
      "ESTOP1_3L+" : ESTOP1;
      "FDBACK_A2.7" : FDBACK;
      "ESTOP1_4L+" : ESTOP1;
      "FDBACK_A2.8" : FDBACK;
      "FDBACK_A2.9" : FDBACK;
      "ESTOP1_5L+" : ESTOP1;
      "F_IEC_Timer_3L+" : TON;
      "F_IEC_Timer_4L+" : TON;
      FDBACK_KF101x : FDBACK;
      FDBACK_KM20_KM21 : FDBACK;
   END_VAR
BEGIN

REGION Network 1: ACK_GL
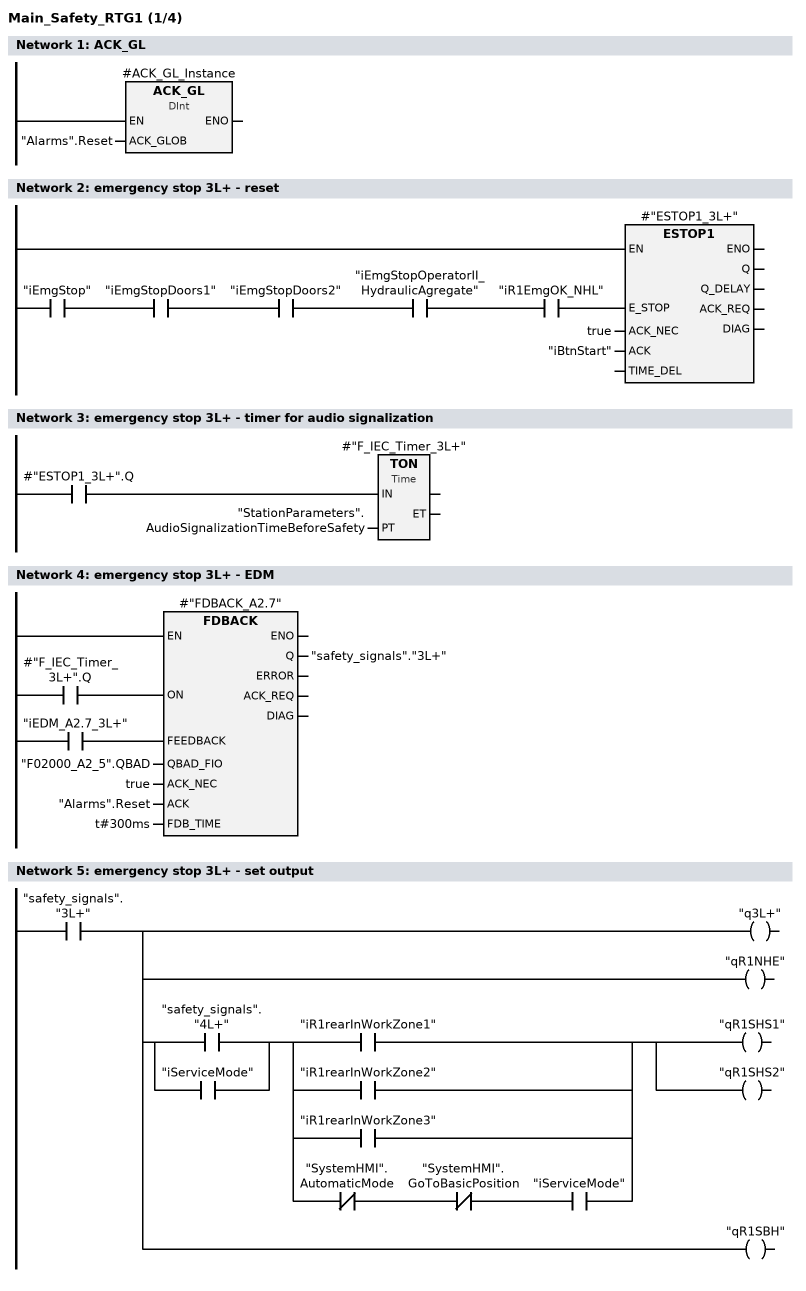
   RUNG wire#powerrail
      { S7_Templates := "codedbool_type := DInt" } #ACK_GL_Instance.ACK_GL(ACK_GLOB := "Alarms".Reset)
   END_RUNG
   // the same network as SCL:
   #ACK_GL_Instance(ACK_GLOB := "Alarms".Reset);   // ACK_GL
END_REGION

REGION Network 2: emergency stop 3L+ - reset
   RUNG wire#powerrail
      #"ESTOP1_3L+".ESTOP1(E_STOP := wire#w1, ACK_NEC := true, ACK := "iBtnStart", TIME_DEL :=, Q =>, Q_DELAY =>, ACK_REQ =>, DIAG =>)
   END_RUNG
   RUNG wire#powerrail
      Contact( "iEmgStop" )
      Contact( "iEmgStopDoors1" )
      Contact( "iEmgStopDoors2" )
      Contact( "iEmgStopOperatorII_HydraulicAgregate" )
      Contact( "iR1EmgOK_NHL" )
   END_RUNG wire#w1
   // the same network as SCL:
   #"ESTOP1_3L+"(E_STOP := "iEmgStop" AND "iEmgStopDoors1" AND "iEmgStopDoors2" AND "iEmgStopOperatorII_HydraulicAgregate" AND "iR1EmgOK_NHL",   // ESTOP1
                 ACK_NEC := true,
                 ACK := "iBtnStart");
END_REGION

REGION Network 3: emergency stop 3L+ - timer for audio signalization
   RUNG wire#powerrail
      Contact( #"ESTOP1_3L+".Q )
      { S7_Templates := "[time_type := Time, codedbool_type := DInt]" } #"F_IEC_Timer_3L+".TON(pt := "StationParameters".AudioSignalizationTimeBeforeSafety, et =>)
   END_RUNG
   // the same network as SCL:
   #"F_IEC_Timer_3L+".TON(IN := #"ESTOP1_3L+".Q, PT := "StationParameters".AudioSignalizationTimeBeforeSafety);
END_REGION

REGION Network 4: emergency stop 3L+ - EDM
   RUNG wire#powerrail
      #"FDBACK_A2.7".FDBACK(ON := wire#w1, FEEDBACK := wire#w2, QBAD_FIO := "F02000_A2_5".QBAD, ACK_NEC := true, ACK := "Alarms".Reset, FDB_TIME := t#300ms, Q => "safety_signals"."3L+", ERROR =>, ACK_REQ =>, DIAG =>)
   END_RUNG
   RUNG wire#powerrail
      Contact( #"F_IEC_Timer_3L+".Q )
   END_RUNG wire#w1
   RUNG wire#powerrail
      Contact( "iEDM_A2.7_3L+" )
   END_RUNG wire#w2
   // the same network as SCL:
   #"FDBACK_A2.7"(ON := #"F_IEC_Timer_3L+".Q,   // FDBACK
                  FEEDBACK := "iEDM_A2.7_3L+",
                  QBAD_FIO := "F02000_A2_5".QBAD,
                  ACK_NEC := true,
                  ACK := "Alarms".Reset,
                  FDB_TIME := t#300ms,
                  Q => "safety_signals"."3L+");
END_REGION

REGION Network 5: emergency stop 3L+ - set output
   RUNG wire#powerrail
      Contact( "safety_signals"."3L+" )
      wire#w1
      Coil( "q3L+" )
   END_RUNG
   RUNG wire#w1
      Coil( "qR1NHE" )
   END_RUNG
   RUNG wire#w1
      Contact( "safety_signals"."4L+" )
      wire#w2
      Contact( "iR1rearInWorkZone1" )
      wire#w3
      Coil( "qR1SHS1" )
   END_RUNG
   RUNG wire#w1
      Contact( "iServiceMode" )
   END_RUNG wire#w2
   RUNG wire#w2
      Contact( "iR1rearInWorkZone2" )
   END_RUNG wire#w3
   RUNG wire#w2
      Contact( "iR1rearInWorkZone3" )
   END_RUNG wire#w3
   RUNG wire#w2
      I_Contact( "SystemHMI".AutomaticMode )
      I_Contact( "SystemHMI".GoToBasicPosition )
      Contact( "iServiceMode" )
   END_RUNG wire#w3
   RUNG wire#w3
      Coil( "qR1SHS2" )
   END_RUNG
   RUNG wire#w1
      Coil( "qR1SBH" )
   END_RUNG
   // the same network as SCL:
   "q3L+" := "safety_signals"."3L+";
   "qR1NHE" := "safety_signals"."3L+";
   "qR1SHS1" := "safety_signals"."3L+" AND ("safety_signals"."4L+" OR "iServiceMode") AND ("iR1rearInWorkZone1" OR "iR1rearInWorkZone2" OR "iR1rearInWorkZone3" OR (NOT "SystemHMI".AutomaticMode AND NOT "SystemHMI".GoToBasicPosition AND "iServiceMode"));
   "qR1SHS2" := "qR1SHS1";
   "qR1SBH" := "safety_signals"."3L+";
END_REGION

REGION Network 6: emergency stop / service doors 4L+ - reset
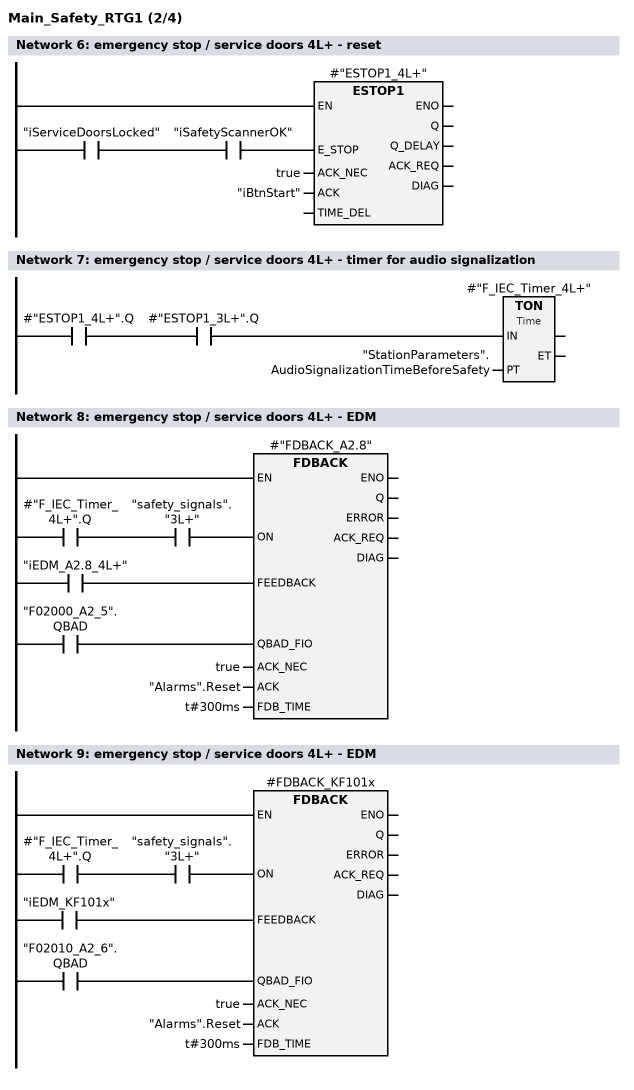
   RUNG wire#powerrail
      #"ESTOP1_4L+".ESTOP1(E_STOP := wire#w1, ACK_NEC := true, ACK := "iBtnStart", TIME_DEL :=, Q =>, Q_DELAY =>, ACK_REQ =>, DIAG =>)
   END_RUNG
   RUNG wire#powerrail
      Contact( "iServiceDoorsLocked" )
      Contact( "iSafetyScannerOK" )
   END_RUNG wire#w1
   // the same network as SCL:
   #"ESTOP1_4L+"(E_STOP := "iServiceDoorsLocked" AND "iSafetyScannerOK", ACK_NEC := true, ACK := "iBtnStart");   // ESTOP1
END_REGION

REGION Network 7: emergency stop / service doors 4L+ - timer for audio signalization
   RUNG wire#powerrail
      Contact( #"ESTOP1_4L+".Q )
      Contact( #"ESTOP1_3L+".Q )
      { S7_Templates := "[time_type := Time, codedbool_type := DInt]" } #"F_IEC_Timer_4L+".TON(pt := "StationParameters".AudioSignalizationTimeBeforeSafety, et =>)
   END_RUNG
   // the same network as SCL:
   #"F_IEC_Timer_4L+".TON(IN := #"ESTOP1_4L+".Q AND #"ESTOP1_3L+".Q,
                          PT := "StationParameters".AudioSignalizationTimeBeforeSafety);
END_REGION

REGION Network 8: emergency stop / service doors 4L+ - EDM
   RUNG wire#powerrail
      #"FDBACK_A2.8".FDBACK(ON := wire#w1, FEEDBACK := wire#w2, QBAD_FIO := wire#w3, ACK_NEC := true, ACK := "Alarms".Reset, FDB_TIME := t#300ms, Q =>, ERROR =>, ACK_REQ =>, DIAG =>)
   END_RUNG
   RUNG wire#powerrail
      Contact( #"F_IEC_Timer_4L+".Q )
      Contact( "safety_signals"."3L+" )
   END_RUNG wire#w1
   RUNG wire#powerrail
      Contact( "iEDM_A2.8_4L+" )
   END_RUNG wire#w2
   RUNG wire#powerrail
      Contact( "F02000_A2_5".QBAD )
   END_RUNG wire#w3
   // the same network as SCL:
   #"FDBACK_A2.8"(ON := #"F_IEC_Timer_4L+".Q AND "safety_signals"."3L+",   // FDBACK
                  FEEDBACK := "iEDM_A2.8_4L+",
                  QBAD_FIO := "F02000_A2_5".QBAD,
                  ACK_NEC := true,
                  ACK := "Alarms".Reset,
                  FDB_TIME := t#300ms);
END_REGION

REGION Network 9: emergency stop / service doors 4L+ - EDM
   RUNG wire#powerrail
      #FDBACK_KF101x.FDBACK(ON := wire#w1, FEEDBACK := wire#w2, QBAD_FIO := wire#w3, ACK_NEC := true, ACK := "Alarms".Reset, FDB_TIME := t#300ms, Q =>, ERROR =>, ACK_REQ =>, DIAG =>)
   END_RUNG
   RUNG wire#powerrail
      Contact( #"F_IEC_Timer_4L+".Q )
      Contact( "safety_signals"."3L+" )
   END_RUNG wire#w1
   RUNG wire#powerrail
      Contact( "iEDM_KF101x" )
   END_RUNG wire#w2
   RUNG wire#powerrail
      Contact( "F02010_A2_6".QBAD )
   END_RUNG wire#w3
   // the same network as SCL:
   #FDBACK_KF101x(ON := #"F_IEC_Timer_4L+".Q AND "safety_signals"."3L+",   // FDBACK
                  FEEDBACK := "iEDM_KF101x",
                  QBAD_FIO := "F02010_A2_6".QBAD,
                  ACK_NEC := true,
                  ACK := "Alarms".Reset,
                  FDB_TIME := t#300ms);
END_REGION

REGION Network 10: emergency stop / service doors 4L+ - set output
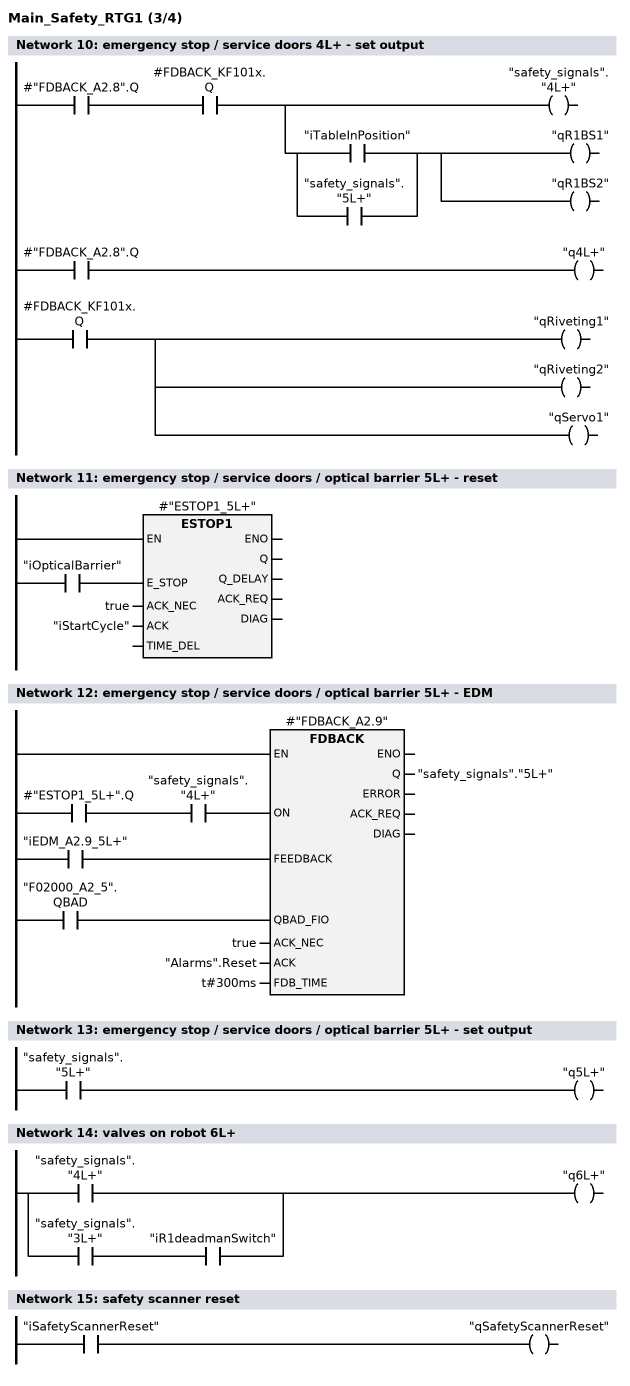
   RUNG wire#powerrail
      Contact( #"FDBACK_A2.8".Q )
      Contact( #FDBACK_KF101x.Q )
      wire#w1
      Coil( "safety_signals"."4L+" )
   END_RUNG
   RUNG wire#w1
      Contact( "iTableInPosition" )
      wire#w2
      Coil( "qR1BS1" )
   END_RUNG
   RUNG wire#w1
      Contact( "safety_signals"."5L+" )
   END_RUNG wire#w2
   RUNG wire#w2
      Coil( "qR1BS2" )
   END_RUNG
   RUNG wire#powerrail
      Contact( #"FDBACK_A2.8".Q )
      Coil( "q4L+" )
   END_RUNG
   RUNG wire#powerrail
      Contact( #FDBACK_KF101x.Q )
      wire#w3
      Coil( "qRiveting1" )
   END_RUNG
   RUNG wire#w3
      Coil( "qRiveting2" )
   END_RUNG
   RUNG wire#w3
      Coil( "qServo1" )
   END_RUNG
   // the same network as SCL:
   "safety_signals"."4L+" := #"FDBACK_A2.8".Q AND #FDBACK_KF101x.Q;
   "qR1BS1" := "safety_signals"."4L+" AND ("iTableInPosition" OR "safety_signals"."5L+");
   "qR1BS2" := "qR1BS1";
   "q4L+" := #"FDBACK_A2.8".Q;
   "qRiveting1" := #FDBACK_KF101x.Q;
   "qRiveting2" := #FDBACK_KF101x.Q;
   "qServo1" := #FDBACK_KF101x.Q;
END_REGION

REGION Network 11: emergency stop / service doors / optical barrier 5L+ - reset
   RUNG wire#powerrail
      #"ESTOP1_5L+".ESTOP1(E_STOP := wire#w1, ACK_NEC := true, ACK := "iStartCycle", TIME_DEL :=, Q =>, Q_DELAY =>, ACK_REQ =>, DIAG =>)
   END_RUNG
   RUNG wire#powerrail
      Contact( "iOpticalBarrier" )
   END_RUNG wire#w1
   // the same network as SCL:
   #"ESTOP1_5L+"(E_STOP := "iOpticalBarrier", ACK_NEC := true, ACK := "iStartCycle");   // ESTOP1
END_REGION

REGION Network 12: emergency stop / service doors / optical barrier 5L+ - EDM
   RUNG wire#powerrail
      #"FDBACK_A2.9".FDBACK(ON := wire#w1, FEEDBACK := wire#w2, QBAD_FIO := wire#w3, ACK_NEC := true, ACK := "Alarms".Reset, FDB_TIME := t#300ms, Q => "safety_signals"."5L+", ERROR =>, ACK_REQ =>, DIAG =>)
   END_RUNG
   RUNG wire#powerrail
      Contact( #"ESTOP1_5L+".Q )
      Contact( "safety_signals"."4L+" )
   END_RUNG wire#w1
   RUNG wire#powerrail
      Contact( "iEDM_A2.9_5L+" )
   END_RUNG wire#w2
   RUNG wire#powerrail
      Contact( "F02000_A2_5".QBAD )
   END_RUNG wire#w3
   // the same network as SCL:
   #"FDBACK_A2.9"(ON := #"ESTOP1_5L+".Q AND "safety_signals"."4L+",   // FDBACK
                  FEEDBACK := "iEDM_A2.9_5L+",
                  QBAD_FIO := "F02000_A2_5".QBAD,
                  ACK_NEC := true,
                  ACK := "Alarms".Reset,
                  FDB_TIME := t#300ms,
                  Q => "safety_signals"."5L+");
END_REGION

REGION Network 13: emergency stop / service doors / optical barrier 5L+ - set output
   RUNG wire#powerrail
      Contact( "safety_signals"."5L+" )
      Coil( "q5L+" )
   END_RUNG
   // the same network as SCL:
   "q5L+" := "safety_signals"."5L+";
END_REGION

REGION Network 14: valves on robot 6L+
   RUNG wire#powerrail
      Contact( "safety_signals"."4L+" )
      wire#w1
      Coil( "q6L+" )
   END_RUNG
   RUNG wire#powerrail
      Contact( "safety_signals"."3L+" )
      Contact( "iR1deadmanSwitch" )
   END_RUNG wire#w1
   // the same network as SCL:
   "q6L+" := "safety_signals"."4L+" OR ("safety_signals"."3L+" AND "iR1deadmanSwitch");
END_REGION

REGION Network 15: safety scanner reset
   RUNG wire#powerrail
      Contact( "iSafetyScannerReset" )
      Coil( "qSafetyScannerReset" )
   END_RUNG
   // the same network as SCL:
   "qSafetyScannerReset" := "iSafetyScannerReset";
END_REGION

REGION Network 16: tool selection for robot - mandatory, but not used
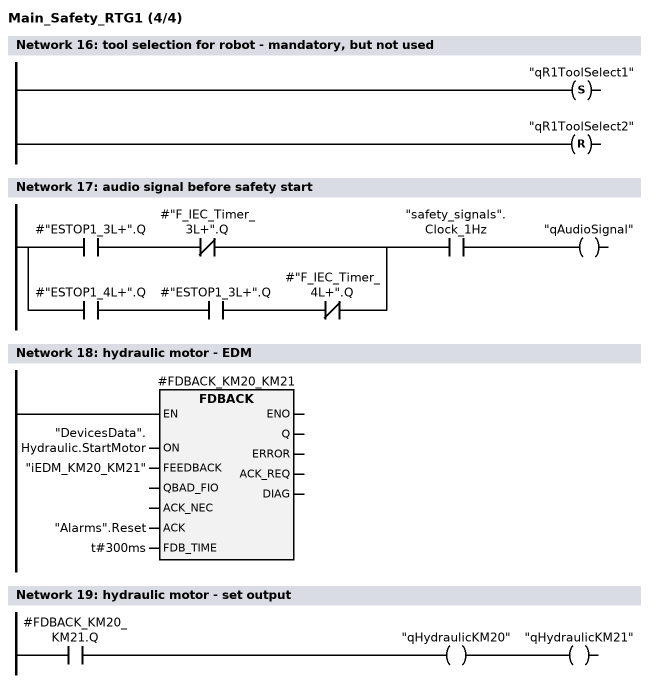
   RUNG wire#powerrail
      S_Coil( "qR1ToolSelect1" )
   END_RUNG
   RUNG wire#powerrail
      R_Coil( "qR1ToolSelect2" )
   END_RUNG
   // the same network as SCL:
   "qR1ToolSelect1" := TRUE;
   "qR1ToolSelect2" := FALSE;
END_REGION

REGION Network 17: audio signal before safety start
   RUNG wire#powerrail
      Contact( #"ESTOP1_3L+".Q )
      I_Contact( #"F_IEC_Timer_3L+".Q )
      wire#w1
      Contact( "safety_signals".Clock_1Hz )
      Coil( "qAudioSignal" )
   END_RUNG
   RUNG wire#powerrail
      Contact( #"ESTOP1_4L+".Q )
      Contact( #"ESTOP1_3L+".Q )
      I_Contact( #"F_IEC_Timer_4L+".Q )
   END_RUNG wire#w1
   // the same network as SCL:
   "qAudioSignal" := ((#"ESTOP1_3L+".Q AND NOT #"F_IEC_Timer_3L+".Q) OR (#"ESTOP1_4L+".Q AND #"ESTOP1_3L+".Q AND NOT #"F_IEC_Timer_4L+".Q)) AND "safety_signals".Clock_1Hz;
END_REGION

REGION Network 18: hydraulic motor - EDM
   RUNG wire#powerrail
      #FDBACK_KM20_KM21.FDBACK(ON := "DevicesData".Hydraulic.StartMotor, FEEDBACK := "iEDM_KM20_KM21", QBAD_FIO :=, ACK_NEC :=, ACK := "Alarms".Reset, FDB_TIME := t#300ms, Q =>, ERROR =>, ACK_REQ =>, DIAG =>)
   END_RUNG
   // the same network as SCL:
   #FDBACK_KM20_KM21(ON := "DevicesData".Hydraulic.StartMotor,   // FDBACK
                     FEEDBACK := "iEDM_KM20_KM21",
                     ACK := "Alarms".Reset,
                     FDB_TIME := t#300ms);
END_REGION

REGION Network 19: hydraulic motor - set output
   RUNG wire#powerrail
      Contact( #FDBACK_KM20_KM21.Q )
      Coil( "qHydraulicKM20" )
      Coil( "qHydraulicKM21" )
   END_RUNG
   // the same network as SCL:
   "qHydraulicKM20" := #FDBACK_KM20_KM21.Q;
   "qHydraulicKM21" := #FDBACK_KM20_KM21.Q;
END_REGION
END_FUNCTION_BLOCK

FUNCTION_BLOCK "sq_autoeject"   // FB53, GRAPH
VERSION : 0.1
// stored: AcknowledgeErrorsRequired true, AutoNumber true, GraphVersion 6.0, InitialValuesAcquisition false, IsIECCheckEnabled false, LanguageInNetworks LAD, LockOperatingMode false, PermanentILProcessingInMANMode false, SetENOAutomatically false, SkipSteps false, UDAEnableTagReadback false, WithAlarmHandling true
   // inherited from GRAPH_BASE
   VAR
      OFF_SQ_BASE : Bool;
   END_VAR
   VAR_INPUT
      OFF_SQ { ExternalWritable := 'False'} : Bool := false;   // Turn sequence off
      INIT_SQ { ExternalWritable := 'False'} : Bool := false;   // Set sequence to initial state
      ACK_EF { ExternalWritable := 'False'} : Bool := false;   // Acknowledge all errors and faults
      S_PREV { ExternalWritable := 'False'} : Bool := false;   // Output previous step in parameter S_NO
      S_NEXT { ExternalWritable := 'False'} : Bool := false;   // Indicate next step in parameter S_NO
      SW_AUTO { ExternalWritable := 'False'} : Bool := false;   // Automatic mode
      SW_TAP { ExternalWritable := 'False'} : Bool := false;   // Semiautomatic/switch with transition
      SW_TOP { ExternalWritable := 'False'} : Bool := false;   // Semiautomatic/ignore transition
      SW_MAN { ExternalWritable := 'False'} : Bool := false;   // Manual mode
      S_SEL { ExternalWritable := 'False'} : Int := 0;   // Select step to be output to S_NO
      S_ON { ExternalWritable := 'False'} : Bool := false;   // Activate step indicated in S_NO
      S_OFF { ExternalWritable := 'False'} : Bool := false;   // Deactivate step indicated S_NO
      T_PUSH { ExternalWritable := 'False'} : Bool := false;   // Enable transition to switch in semi automatic mode
   END_VAR
   VAR_OUTPUT
      S_NO { ExternalWritable := 'False'} : Int := 0;   // Step number
      S_MORE { ExternalWritable := 'False'} : Bool := false;   // More steps are available and can be shown in S_NO
      S_ACTIVE { ExternalWritable := 'False'} : Bool := false;   // Step indicated in S_NO is active
      ERR_FLT { ExternalWritable := 'False'} : Bool := false;   // Interlock or supervision group error
      AUTO_ON { ExternalWritable := 'False'} : Bool := false;   // Automatic mode is active
      TAP_ON { ExternalWritable := 'False'} : Bool := false;   // Semiautomatic mode/step with transition enabled
      TOP_ON { ExternalWritable := 'False'} : Bool := false;   // Semiautomatic mode/ignore transition enabled
      MAN_ON { ExternalWritable := 'False'} : Bool := false;   // Manual mode is active
   END_VAR
   VAR
      dummy : Bool;
      start : Bool;
      base : Bool;
   END_VAR
BEGIN
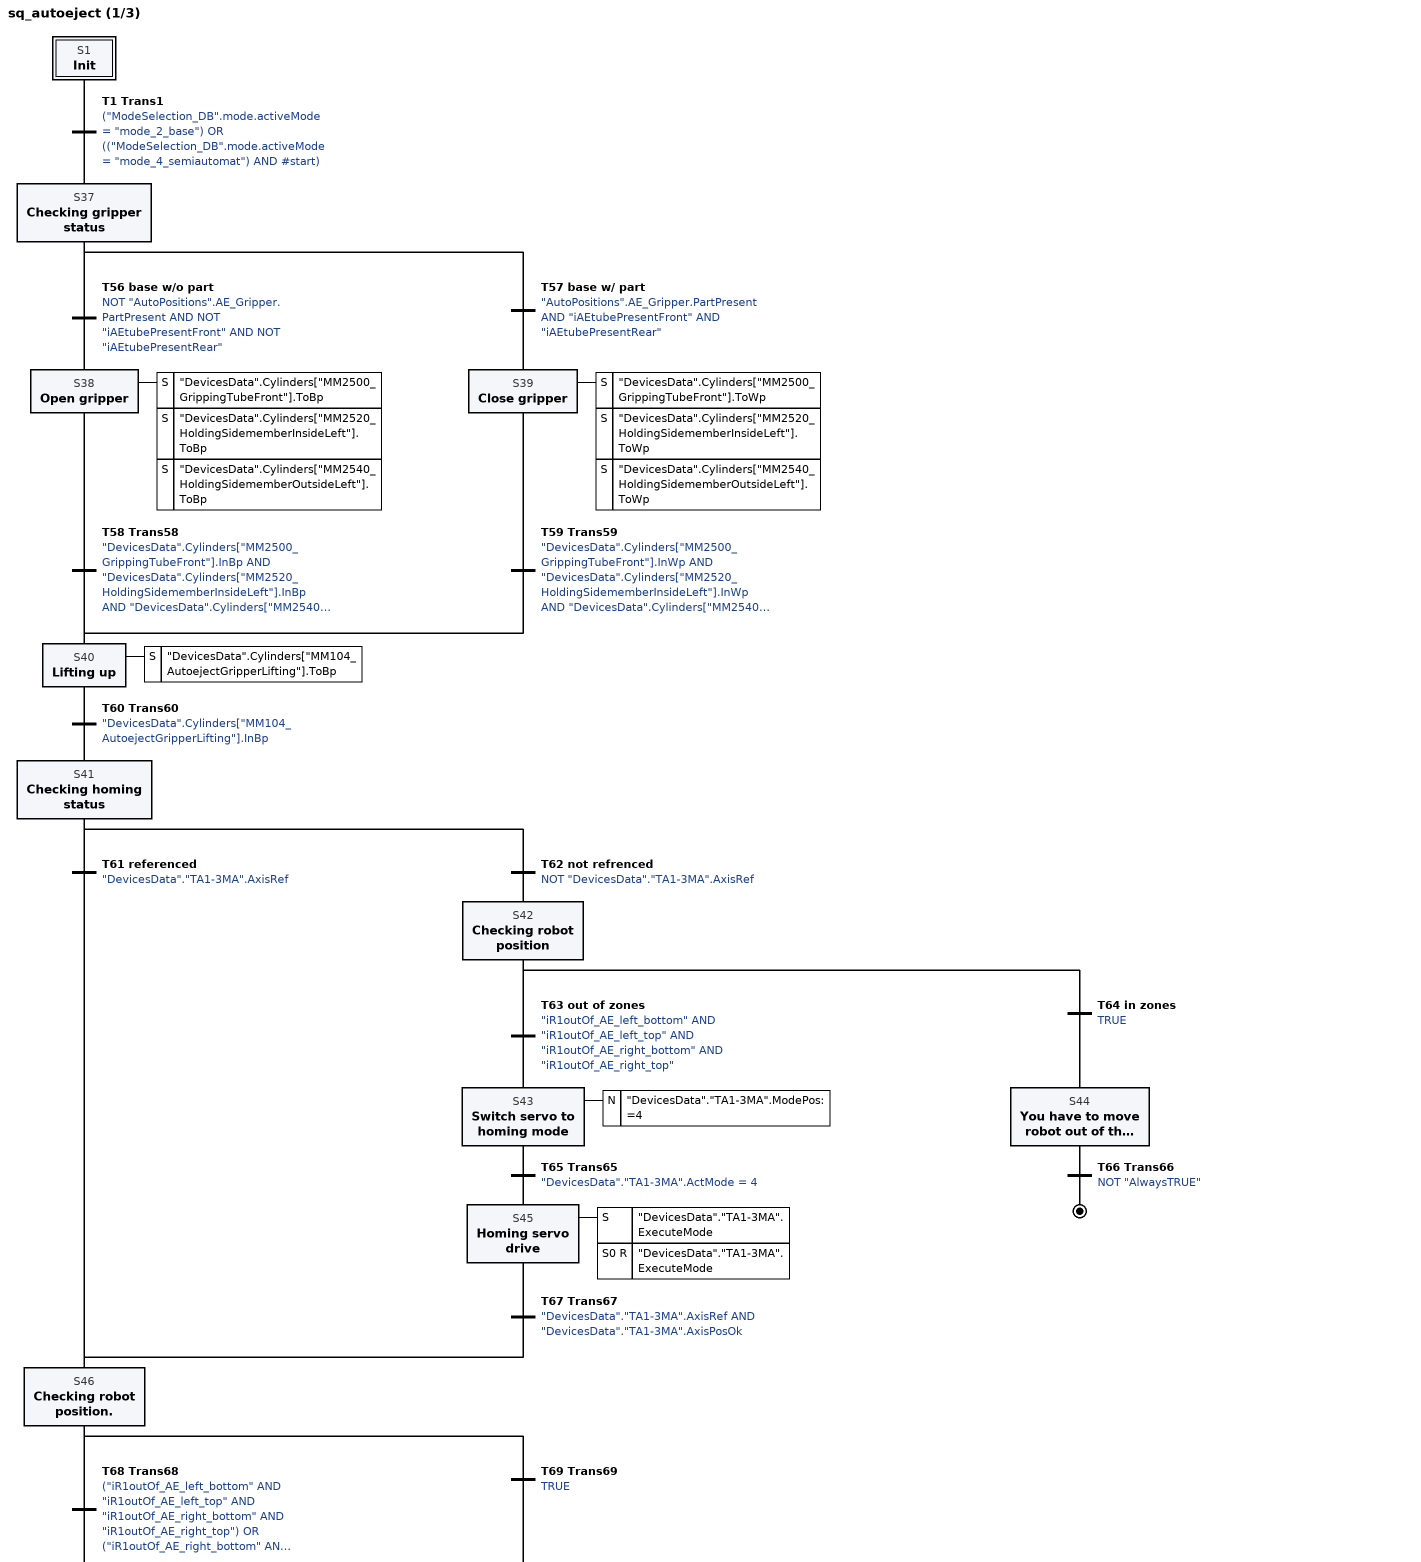
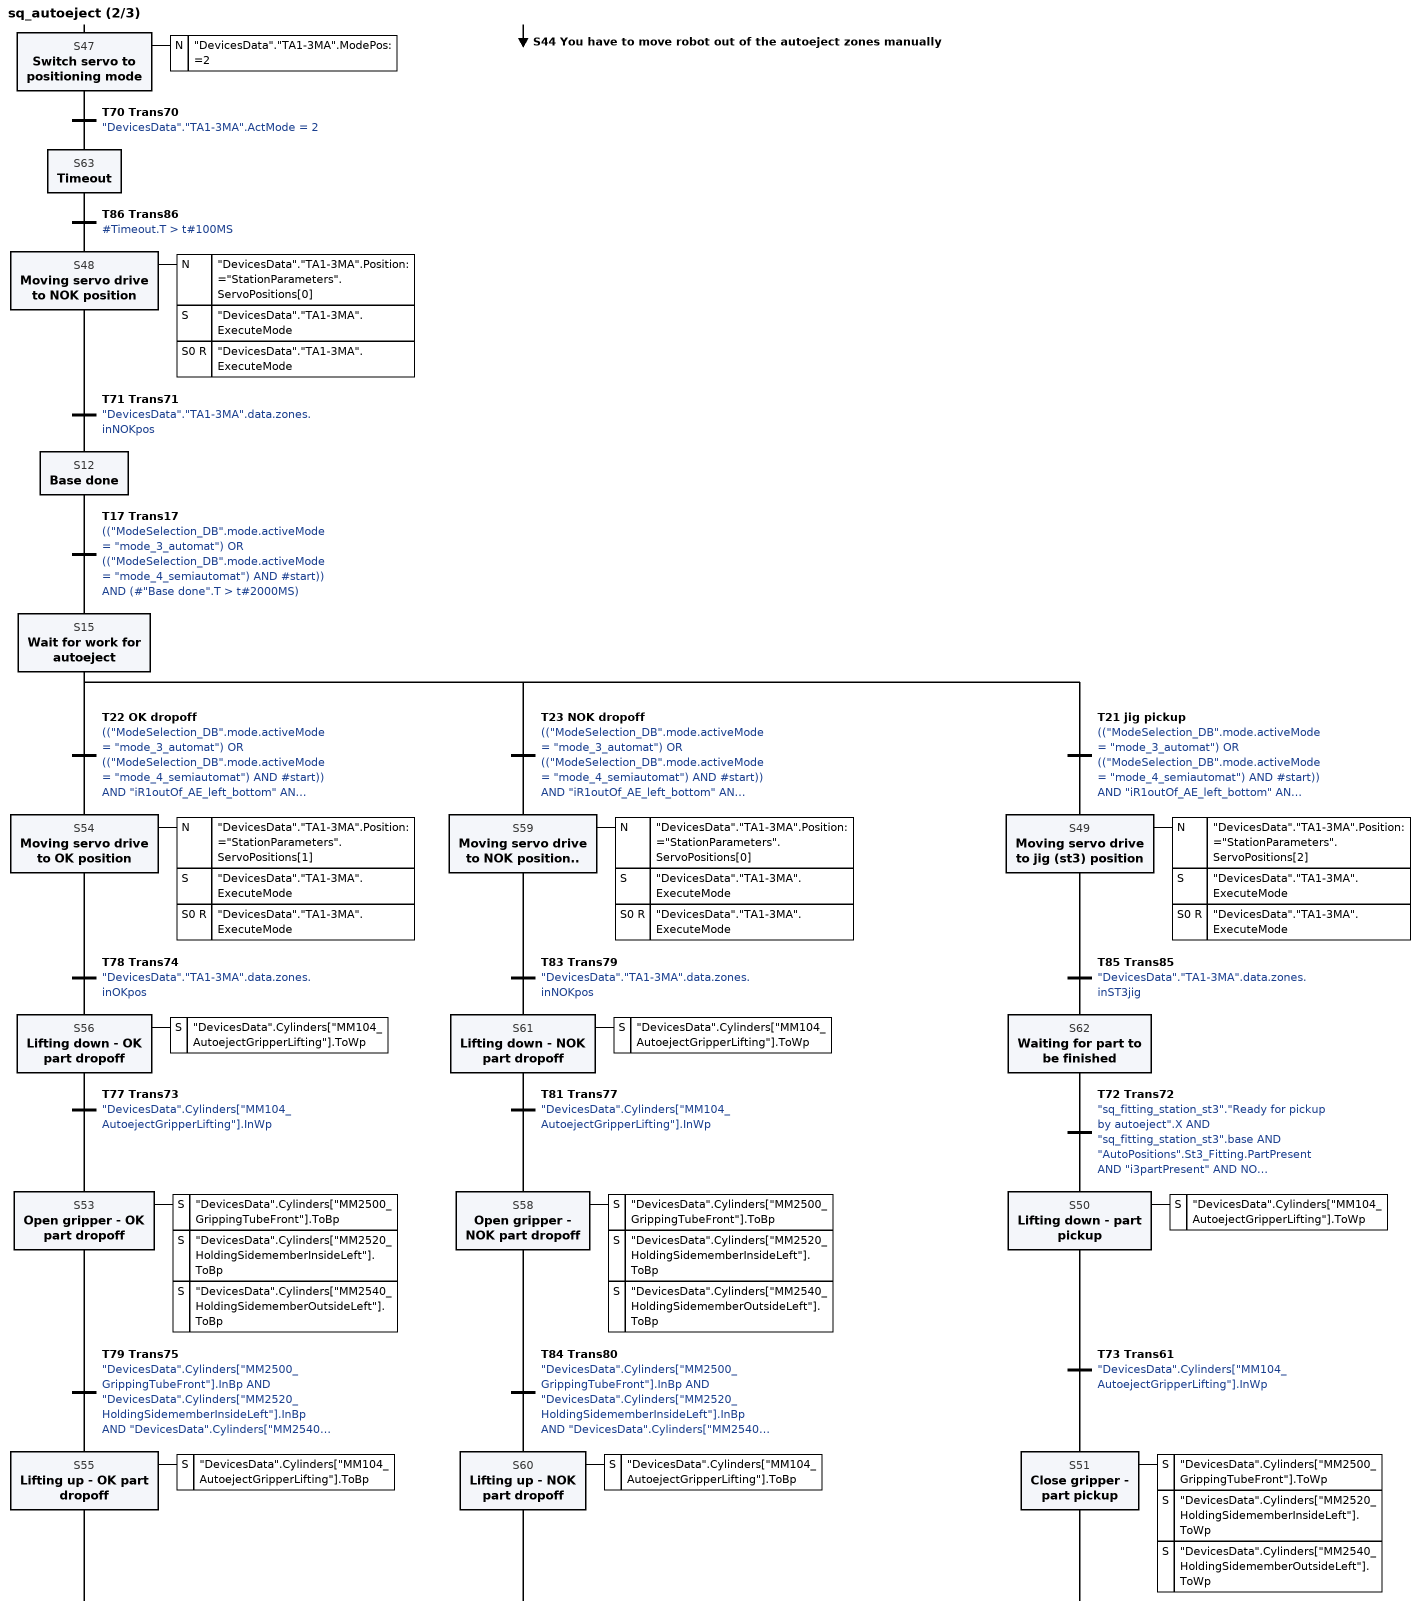
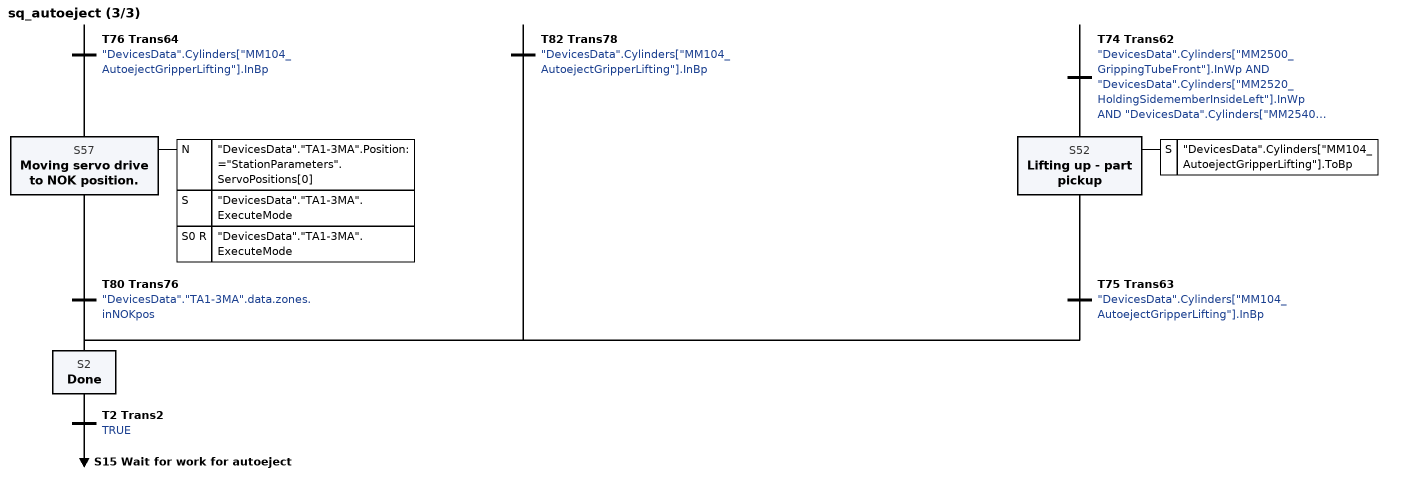
   // sequencer 1
   INITIAL_STEP Init:   // S1, max time T#10S, warning time T#7S
   END_STEP
   TRANSITION Trans1 FROM Init TO "Checking gripper status"   // T1
      := ("ModeSelection_DB".mode.activeMode = "mode_2_base") OR (("ModeSelection_DB".mode.activeMode = "mode_4_semiautomat") AND #start);
   END_TRANSITION
   STEP Done:   // S2, max time T#10S, warning time T#7S
   END_STEP
   TRANSITION Trans2 FROM Done TO "Wait for work for autoeject"   // T2, jump
      := TRUE;
   END_TRANSITION
   STEP "Base done":   // S12, max time T#10S, warning time T#7S
   END_STEP
   TRANSITION Trans17 FROM "Base done" TO "Wait for work for autoeject"   // T17
      := (("ModeSelection_DB".mode.activeMode = "mode_3_automat") OR (("ModeSelection_DB".mode.activeMode = "mode_4_semiautomat") AND #start)) AND (#"Base done".T > t#2000MS);
   END_TRANSITION
   STEP "Wait for work for autoeject":   // S15, max time T#10S, warning time T#7S
   END_STEP
   TRANSITION "OK dropoff" FROM "Wait for work for autoeject" TO "Moving servo drive to OK position"   // T22
      := (("ModeSelection_DB".mode.activeMode = "mode_3_automat") OR (("ModeSelection_DB".mode.activeMode = "mode_4_semiautomat") AND #start)) AND "iR1outOf_AE_left_bottom" AND "iR1outOf_AE_left_top" AND "iR1outOf_AE_right_bottom" AND "iR1outOf_AE_right_top" AND "AutoPositions".AE_Gripper.PartPresent AND "AutoPositions".AE_Gripper.StFinished[3] AND NOT "AutoPositions".AE_Gripper.PartNOK AND "iAEtubePresentFront" AND "iAEtubePresentRear" AND NOT "AutoPositions".St4_OKposition.PartPresent AND NOT "i4partPresent";
   END_TRANSITION
   TRANSITION "NOK dropoff" FROM "Wait for work for autoeject" TO "Moving servo drive to NOK position.."   // T23
      := (("ModeSelection_DB".mode.activeMode = "mode_3_automat") OR (("ModeSelection_DB".mode.activeMode = "mode_4_semiautomat") AND #start)) AND "iR1outOf_AE_left_bottom" AND "iR1outOf_AE_left_top" AND "iR1outOf_AE_right_bottom" AND "iR1outOf_AE_right_top" AND "AutoPositions".AE_Gripper.PartPresent AND (NOT "AutoPositions".AE_Gripper.StFinished[3] OR "AutoPositions".AE_Gripper.PartNOK) AND "iAEtubePresentFront" AND "iAEtubePresentRear" AND NOT "PartHolderData".NOKBoxFull;
   END_TRANSITION
   TRANSITION "jig pickup" FROM "Wait for work for autoeject" TO "Moving servo drive to jig (st3) position"   // T21
      := (("ModeSelection_DB".mode.activeMode = "mode_3_automat") OR (("ModeSelection_DB".mode.activeMode = "mode_4_semiautomat") AND #start)) AND "iR1outOf_AE_left_bottom" AND "iR1outOf_AE_left_top" AND "iR1outOf_AE_right_bottom" AND "iR1outOf_AE_right_top" AND "AutoPositions".St3_Fitting.PartPresent AND "i3partPresent" AND NOT "AutoPositions".AE_Gripper.PartPresent AND NOT "iAEtubePresentFront" AND NOT "iAEtubePresentRear" AND NOT "AutoPositions".St4_OKposition.PartPresent AND NOT "i4partPresent";
   END_TRANSITION
   STEP "Close gripper - part pickup":   // S51, max time T#10S, warning time T#7S
              S    "DevicesData".Cylinders["MM2500_GrippingTubeFront"].ToWp
              S    "DevicesData".Cylinders["MM2520_HoldingSidememberInsideLeft"].ToWp
              S    "DevicesData".Cylinders["MM2540_HoldingSidememberOutsideLeft"].ToWp
   END_STEP
   TRANSITION Trans62 FROM "Close gripper - part pickup" TO "Lifting up - part pickup"   // T74
      := "DevicesData".Cylinders["MM2500_GrippingTubeFront"].InWp AND "DevicesData".Cylinders["MM2520_HoldingSidememberInsideLeft"].InWp AND "DevicesData".Cylinders["MM2540_HoldingSidememberOutsideLeft"].InWp;
   END_TRANSITION
   STEP "Open gripper - OK part dropoff":   // S53, max time T#10S, warning time T#7S
              S    "DevicesData".Cylinders["MM2500_GrippingTubeFront"].ToBp
              S    "DevicesData".Cylinders["MM2520_HoldingSidememberInsideLeft"].ToBp
              S    "DevicesData".Cylinders["MM2540_HoldingSidememberOutsideLeft"].ToBp
   END_STEP
   TRANSITION Trans75 FROM "Open gripper - OK part dropoff" TO "Lifting up - OK part dropoff"   // T79
      := "DevicesData".Cylinders["MM2500_GrippingTubeFront"].InBp AND "DevicesData".Cylinders["MM2520_HoldingSidememberInsideLeft"].InBp AND "DevicesData".Cylinders["MM2540_HoldingSidememberOutsideLeft"].InBp;
   END_TRANSITION
   STEP "Moving servo drive to OK position":   // S54, max time T#30S, warning time T#7S
      supervision V := #"Moving servo drive to OK position".T > #"Moving servo drive to OK position".T_MAX;
              N    "DevicesData"."TA1-3MA".Position:="StationParameters".ServoPositions[1]
              S    "DevicesData"."TA1-3MA".ExecuteMode
          S0  R    "DevicesData"."TA1-3MA".ExecuteMode
   END_STEP
   TRANSITION Trans74 FROM "Moving servo drive to OK position" TO "Lifting down - OK part dropoff"   // T78
      := "DevicesData"."TA1-3MA".data.zones.inOKpos;
   END_TRANSITION
   STEP "Lifting up - OK part dropoff":   // S55, max time T#10S, warning time T#7S
              S    "DevicesData".Cylinders["MM104_AutoejectGripperLifting"].ToBp
   END_STEP
   TRANSITION Trans64 FROM "Lifting up - OK part dropoff" TO "Moving servo drive to NOK position."   // T76
      := "DevicesData".Cylinders["MM104_AutoejectGripperLifting"].InBp;
   END_TRANSITION
   STEP "Lifting down - OK part dropoff":   // S56, max time T#10S, warning time T#7S
              S    "DevicesData".Cylinders["MM104_AutoejectGripperLifting"].ToWp
   END_STEP
   TRANSITION Trans73 FROM "Lifting down - OK part dropoff" TO "Open gripper - OK part dropoff"   // T77
      := "DevicesData".Cylinders["MM104_AutoejectGripperLifting"].InWp;
   END_TRANSITION
   STEP "Moving servo drive to jig (st3) position":   // S49, max time T#30S, warning time T#7S
      supervision V := #"Moving servo drive to jig (st3) position".T > #"Moving servo drive to jig (st3) position".T_MAX;
              N    "DevicesData"."TA1-3MA".Position:="StationParameters".ServoPositions[2]
              S    "DevicesData"."TA1-3MA".ExecuteMode
          S0  R    "DevicesData"."TA1-3MA".ExecuteMode
   END_STEP
   TRANSITION Trans85 FROM "Moving servo drive to jig (st3) position" TO "Waiting for part to be finished"   // T85
      := "DevicesData"."TA1-3MA".data.zones.inST3jig;
   END_TRANSITION
   STEP "Lifting up - part pickup":   // S52, max time T#10S, warning time T#7S
              S    "DevicesData".Cylinders["MM104_AutoejectGripperLifting"].ToBp
   END_STEP
   TRANSITION Trans63 FROM "Lifting up - part pickup" TO Done   // T75
      := "DevicesData".Cylinders["MM104_AutoejectGripperLifting"].InBp;
   END_TRANSITION
   STEP "Lifting down - part pickup":   // S50, max time T#10S, warning time T#7S
              S    "DevicesData".Cylinders["MM104_AutoejectGripperLifting"].ToWp
   END_STEP
   TRANSITION Trans61 FROM "Lifting down - part pickup" TO "Close gripper - part pickup"   // T73
      := "DevicesData".Cylinders["MM104_AutoejectGripperLifting"].InWp;
   END_TRANSITION
   STEP "Checking gripper status":   // S37, max time T#10S, warning time T#7S
   END_STEP
   TRANSITION "base w/o part" FROM "Checking gripper status" TO "Open gripper"   // T56
      := NOT "AutoPositions".AE_Gripper.PartPresent AND NOT "iAEtubePresentFront" AND NOT "iAEtubePresentRear";
   END_TRANSITION
   TRANSITION "base w/ part" FROM "Checking gripper status" TO "Close gripper"   // T57
      := "AutoPositions".AE_Gripper.PartPresent AND "iAEtubePresentFront" AND "iAEtubePresentRear";
   END_TRANSITION
   STEP "Open gripper":   // S38, max time T#10S, warning time T#7S
              S    "DevicesData".Cylinders["MM2500_GrippingTubeFront"].ToBp
              S    "DevicesData".Cylinders["MM2520_HoldingSidememberInsideLeft"].ToBp
              S    "DevicesData".Cylinders["MM2540_HoldingSidememberOutsideLeft"].ToBp
   END_STEP
   TRANSITION Trans58 FROM "Open gripper" TO "Lifting up"   // T58
      := "DevicesData".Cylinders["MM2500_GrippingTubeFront"].InBp AND "DevicesData".Cylinders["MM2520_HoldingSidememberInsideLeft"].InBp AND "DevicesData".Cylinders["MM2540_HoldingSidememberOutsideLeft"].InBp;
   END_TRANSITION
   STEP "Close gripper":   // S39, max time T#10S, warning time T#7S
              S    "DevicesData".Cylinders["MM2500_GrippingTubeFront"].ToWp
              S    "DevicesData".Cylinders["MM2520_HoldingSidememberInsideLeft"].ToWp
              S    "DevicesData".Cylinders["MM2540_HoldingSidememberOutsideLeft"].ToWp
   END_STEP
   TRANSITION Trans59 FROM "Close gripper" TO "Lifting up"   // T59
      := "DevicesData".Cylinders["MM2500_GrippingTubeFront"].InWp AND "DevicesData".Cylinders["MM2520_HoldingSidememberInsideLeft"].InWp AND "DevicesData".Cylinders["MM2540_HoldingSidememberOutsideLeft"].InWp;
   END_TRANSITION
   STEP "Lifting up":   // S40, max time T#10S, warning time T#7S
              S    "DevicesData".Cylinders["MM104_AutoejectGripperLifting"].ToBp
   END_STEP
   TRANSITION Trans60 FROM "Lifting up" TO "Checking homing status"   // T60
      := "DevicesData".Cylinders["MM104_AutoejectGripperLifting"].InBp;
   END_TRANSITION
   STEP "Checking homing status":   // S41, max time T#10S, warning time T#7S
   END_STEP
   TRANSITION referenced FROM "Checking homing status" TO "Checking robot position."   // T61
      := "DevicesData"."TA1-3MA".AxisRef;
   END_TRANSITION
   TRANSITION "not refrenced" FROM "Checking homing status" TO "Checking robot position"   // T62
      := NOT "DevicesData"."TA1-3MA".AxisRef;
   END_TRANSITION
   STEP "Checking robot position":   // S42, max time T#10S, warning time T#7S
   END_STEP
   TRANSITION "out of zones" FROM "Checking robot position" TO "Switch servo to homing mode"   // T63
      := "iR1outOf_AE_left_bottom" AND "iR1outOf_AE_left_top" AND "iR1outOf_AE_right_bottom" AND "iR1outOf_AE_right_top";
   END_TRANSITION
   TRANSITION "in zones" FROM "Checking robot position" TO "You have to move robot out of the autoeject zones manually"   // T64
      := TRUE;
   END_TRANSITION
   STEP "Switch servo to homing mode":   // S43, max time T#10S, warning time T#7S
      supervision V := #"Switch servo to homing mode".T > #"Switch servo to homing mode".T_MAX;
              N    "DevicesData"."TA1-3MA".ModePos:=4
   END_STEP
   TRANSITION Trans65 FROM "Switch servo to homing mode" TO "Homing servo drive"   // T65
      := "DevicesData"."TA1-3MA".ActMode = 4;
   END_TRANSITION
   STEP "You have to move robot out of the autoeject zones manually":   // S44, max time T#10S, warning time T#7S
      supervision V := "AlwaysTRUE";
   END_STEP
   TRANSITION Trans66 FROM "You have to move robot out of the autoeject zones manually" TO END   // T66
      := NOT "AlwaysTRUE";
   END_TRANSITION
   STEP "Homing servo drive":   // S45, max time T#30S, warning time T#7S
      supervision V := #"Homing servo drive".T > #"Homing servo drive".T_MAX;
              S    "DevicesData"."TA1-3MA".ExecuteMode
          S0  R    "DevicesData"."TA1-3MA".ExecuteMode
   END_STEP
   TRANSITION Trans67 FROM "Homing servo drive" TO "Checking robot position."   // T67
      := "DevicesData"."TA1-3MA".AxisRef AND "DevicesData"."TA1-3MA".AxisPosOk;
   END_TRANSITION
   STEP "Checking robot position.":   // S46, max time T#10S, warning time T#7S
   END_STEP
   TRANSITION Trans68 FROM "Checking robot position." TO "Switch servo to positioning mode"   // T68
      := ("iR1outOf_AE_left_bottom" AND "iR1outOf_AE_left_top" AND "iR1outOf_AE_right_bottom" AND "iR1outOf_AE_right_top") OR ("iR1outOf_AE_right_bottom" AND "iR1outOf_AE_right_top" AND "DevicesData"."TA1-3MA".data.zones.outOfST3zone);
   END_TRANSITION
   TRANSITION Trans69 FROM "Checking robot position." TO "You have to move robot out of the autoeject zones manually"   // T69, jump
      := TRUE;
   END_TRANSITION
   STEP "Switch servo to positioning mode":   // S47, max time T#10S, warning time T#7S
      supervision V := #"Switch servo to positioning mode".T > #"Switch servo to positioning mode".T_MAX;
              N    "DevicesData"."TA1-3MA".ModePos:=2
   END_STEP
   TRANSITION Trans70 FROM "Switch servo to positioning mode" TO Timeout   // T70
      := "DevicesData"."TA1-3MA".ActMode = 2;
   END_TRANSITION
   STEP "Moving servo drive to NOK position":   // S48, max time T#30S, warning time T#7S
      supervision V := #"Moving servo drive to NOK position".T > #"Moving servo drive to NOK position".T_MAX;
              N    "DevicesData"."TA1-3MA".Position:="StationParameters".ServoPositions[0]
              S    "DevicesData"."TA1-3MA".ExecuteMode
          S0  R    "DevicesData"."TA1-3MA".ExecuteMode
   END_STEP
   TRANSITION Trans71 FROM "Moving servo drive to NOK position" TO "Base done"   // T71
      := "DevicesData"."TA1-3MA".data.zones.inNOKpos;
   END_TRANSITION
   STEP "Moving servo drive to NOK position.":   // S57, max time T#30S, warning time T#7S
      supervision V := #"Moving servo drive to NOK position.".T > #"Moving servo drive to NOK position.".T_MAX;
              N    "DevicesData"."TA1-3MA".Position:="StationParameters".ServoPositions[0]
              S    "DevicesData"."TA1-3MA".ExecuteMode
          S0  R    "DevicesData"."TA1-3MA".ExecuteMode
   END_STEP
   TRANSITION Trans76 FROM "Moving servo drive to NOK position." TO Done   // T80
      := "DevicesData"."TA1-3MA".data.zones.inNOKpos;
   END_TRANSITION
   STEP "Open gripper - NOK part dropoff":   // S58, max time T#10S, warning time T#7S
              S    "DevicesData".Cylinders["MM2500_GrippingTubeFront"].ToBp
              S    "DevicesData".Cylinders["MM2520_HoldingSidememberInsideLeft"].ToBp
              S    "DevicesData".Cylinders["MM2540_HoldingSidememberOutsideLeft"].ToBp
   END_STEP
   TRANSITION Trans80 FROM "Open gripper - NOK part dropoff" TO "Lifting up - NOK part dropoff"   // T84
      := "DevicesData".Cylinders["MM2500_GrippingTubeFront"].InBp AND "DevicesData".Cylinders["MM2520_HoldingSidememberInsideLeft"].InBp AND "DevicesData".Cylinders["MM2540_HoldingSidememberOutsideLeft"].InBp;
   END_TRANSITION
   STEP "Moving servo drive to NOK position..":   // S59, max time T#30S, warning time T#7S
      supervision V := #"Moving servo drive to NOK position..".T > #"Moving servo drive to NOK position..".T_MAX;
              N    "DevicesData"."TA1-3MA".Position:="StationParameters".ServoPositions[0]
              S    "DevicesData"."TA1-3MA".ExecuteMode
          S0  R    "DevicesData"."TA1-3MA".ExecuteMode
   END_STEP
   TRANSITION Trans79 FROM "Moving servo drive to NOK position.." TO "Lifting down - NOK part dropoff"   // T83
      := "DevicesData"."TA1-3MA".data.zones.inNOKpos;
   END_TRANSITION
   STEP "Lifting up - NOK part dropoff":   // S60, max time T#10S, warning time T#7S
              S    "DevicesData".Cylinders["MM104_AutoejectGripperLifting"].ToBp
   END_STEP
   TRANSITION Trans78 FROM "Lifting up - NOK part dropoff" TO Done   // T82
      := "DevicesData".Cylinders["MM104_AutoejectGripperLifting"].InBp;
   END_TRANSITION
   STEP "Lifting down - NOK part dropoff":   // S61, max time T#10S, warning time T#7S
              S    "DevicesData".Cylinders["MM104_AutoejectGripperLifting"].ToWp
   END_STEP
   TRANSITION Trans77 FROM "Lifting down - NOK part dropoff" TO "Open gripper - NOK part dropoff"   // T81
      := "DevicesData".Cylinders["MM104_AutoejectGripperLifting"].InWp;
   END_TRANSITION
   STEP "Waiting for part to be finished":   // S62, max time T#10S, warning time T#7S
   END_STEP
   TRANSITION Trans72 FROM "Waiting for part to be finished" TO "Lifting down - part pickup"   // T72
      := "sq_fitting_station_st3"."Ready for pickup by autoeject".X AND "sq_fitting_station_st3".base AND "AutoPositions".St3_Fitting.PartPresent AND "i3partPresent" AND NOT "AutoPositions".AE_Gripper.PartPresent AND NOT "iAEtubePresentFront" AND NOT "iAEtubePresentRear" AND NOT "AutoPositions".St4_OKposition.PartPresent;
   END_TRANSITION
   STEP Timeout:   // S63, max time T#10S, warning time T#7S
   END_STEP
   TRANSITION Trans86 FROM Timeout TO "Moving servo drive to NOK position"   // T86
      := #Timeout.T > t#100MS;
   END_TRANSITION
END_FUNCTION_BLOCK

FUNCTION_BLOCK "sq_carousel_main"   // FB70, GRAPH
VERSION : 0.1
// stored: AcknowledgeErrorsRequired true, AutoNumber true, GraphVersion 6.0, InitialValuesAcquisition false, IsIECCheckEnabled false, LanguageInNetworks LAD, LockOperatingMode false, PermanentILProcessingInMANMode false, SetENOAutomatically false, SkipSteps false, UDAEnableTagReadback false, WithAlarmHandling true
   // inherited from GRAPH_BASE
   VAR
      OFF_SQ_BASE : Bool;
   END_VAR
   VAR_INPUT
      OFF_SQ { ExternalAccessible := 'False'; ExternalVisible := 'False'; ExternalWritable := 'False'} : Bool := false;   // Turn sequence off
      INIT_SQ { ExternalAccessible := 'False'; ExternalVisible := 'False'; ExternalWritable := 'False'} : Bool := false;   // Set sequence to initial state
      ACK_EF { ExternalAccessible := 'False'; ExternalVisible := 'False'; ExternalWritable := 'False'} : Bool := false;   // Acknowledge all errors and faults
      S_PREV { ExternalAccessible := 'False'; ExternalVisible := 'False'; ExternalWritable := 'False'} : Bool := false;   // Output previous step in parameter S_NO
      S_NEXT { ExternalAccessible := 'False'; ExternalVisible := 'False'; ExternalWritable := 'False'} : Bool := false;   // Indicate next step in parameter S_NO
      SW_AUTO { ExternalAccessible := 'False'; ExternalVisible := 'False'; ExternalWritable := 'False'} : Bool := false;   // Automatic mode
      SW_TAP { ExternalAccessible := 'False'; ExternalVisible := 'False'; ExternalWritable := 'False'} : Bool := false;   // Semiautomatic/switch with transition
      SW_TOP { ExternalAccessible := 'False'; ExternalVisible := 'False'; ExternalWritable := 'False'} : Bool := false;   // Semiautomatic/ignore transition
      SW_MAN { ExternalAccessible := 'False'; ExternalVisible := 'False'; ExternalWritable := 'False'} : Bool := false;   // Manual mode
      S_SEL { ExternalAccessible := 'False'; ExternalVisible := 'False'; ExternalWritable := 'False'} : Int := 0;   // Select step to be output to S_NO
      S_ON { ExternalAccessible := 'False'; ExternalVisible := 'False'; ExternalWritable := 'False'} : Bool := false;   // Activate step indicated in S_NO
      S_OFF { ExternalAccessible := 'False'; ExternalVisible := 'False'; ExternalWritable := 'False'} : Bool := false;   // Deactivate step indicated S_NO
      T_PUSH { ExternalAccessible := 'False'; ExternalVisible := 'False'; ExternalWritable := 'False'} : Bool := false;   // Enable transition to switch in semi automatic mode
   END_VAR
   VAR_OUTPUT
      S_NO { ExternalAccessible := 'False'; ExternalVisible := 'False'; ExternalWritable := 'False'} : Int := 0;   // Step number
      S_MORE { ExternalAccessible := 'False'; ExternalVisible := 'False'; ExternalWritable := 'False'} : Bool := false;   // More steps are available and can be shown in S_NO
      S_ACTIVE { ExternalAccessible := 'False'; ExternalVisible := 'False'; ExternalWritable := 'False'} : Bool := false;   // Step indicated in S_NO is active
      ERR_FLT { ExternalAccessible := 'False'; ExternalVisible := 'False'; ExternalWritable := 'False'} : Bool := false;   // Interlock or supervision group error
      AUTO_ON { ExternalAccessible := 'False'; ExternalVisible := 'False'; ExternalWritable := 'False'} : Bool := false;   // Automatic mode is active
      TAP_ON { ExternalAccessible := 'False'; ExternalVisible := 'False'; ExternalWritable := 'False'} : Bool := false;   // Semiautomatic mode/step with transition enabled
      TOP_ON { ExternalAccessible := 'False'; ExternalVisible := 'False'; ExternalWritable := 'False'} : Bool := false;   // Semiautomatic mode/ignore transition enabled
      MAN_ON { ExternalAccessible := 'False'; ExternalVisible := 'False'; ExternalWritable := 'False'} : Bool := false;   // Manual mode is active
   END_VAR
   VAR
      dummy : Bool;
      start : Bool;
      base : Bool;
   END_VAR
BEGIN
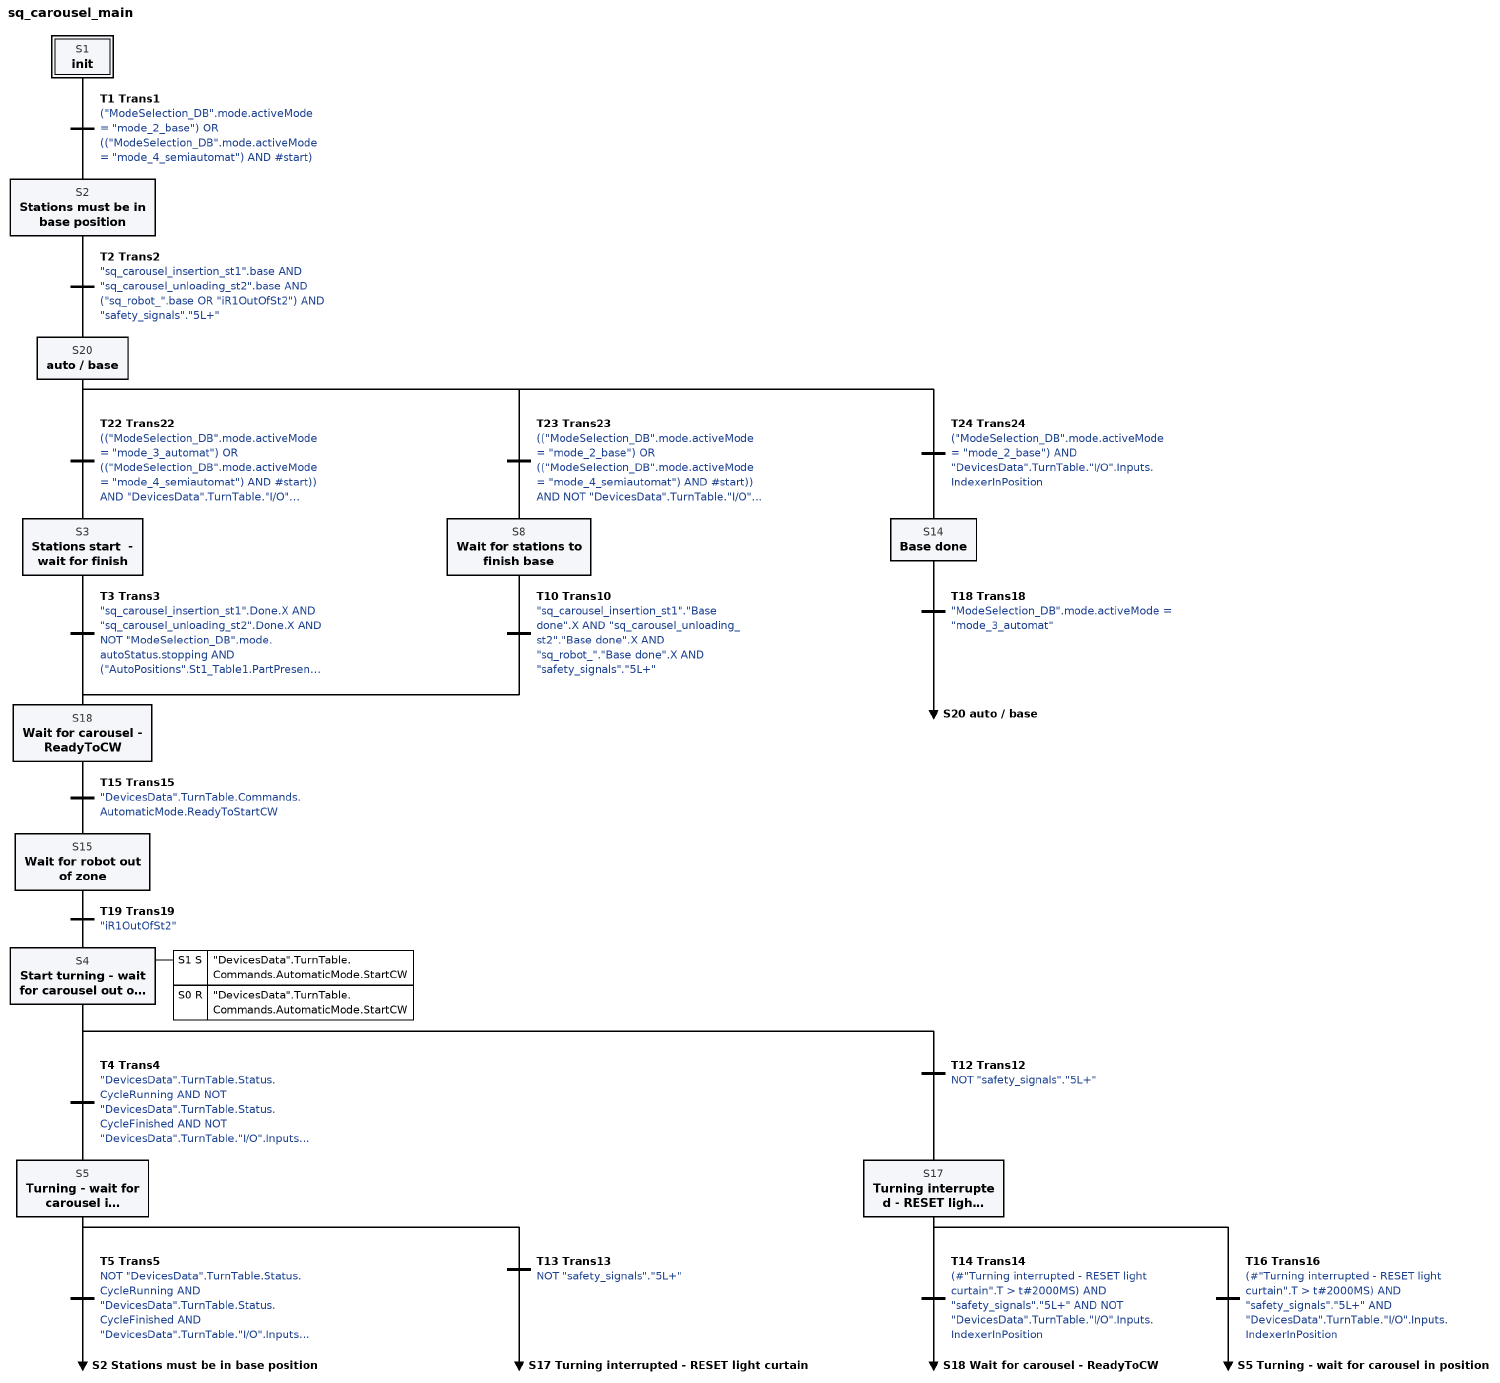
   // permanent pre-instructions
   NETWORK 1
      #base := "iTurnTableIndexerInPosition";

   // sequencer 1
   INITIAL_STEP init:   // S1, max time T#10S, warning time T#7S
   END_STEP
   TRANSITION Trans1 FROM init TO "Stations must be in base position"   // T1
      := ("ModeSelection_DB".mode.activeMode = "mode_2_base") OR (("ModeSelection_DB".mode.activeMode = "mode_4_semiautomat") AND #start);
   END_TRANSITION
   STEP "Stations must be in base position":   // S2, max time T#10S, warning time T#7S
      supervision V := #"Stations must be in base position".T > #"Stations must be in base position".T_MAX;
   END_STEP
   TRANSITION Trans2 FROM "Stations must be in base position" TO "auto / base"   // T2
      := "sq_carousel_insertion_st1".base AND "sq_carousel_unloading_st2".base AND ("sq_robot_".base OR "iR1OutOfSt2") AND "safety_signals"."5L+";
   END_TRANSITION
   STEP "Stations start  - wait for finish":   // S3, max time T#10S, warning time T#7S
   END_STEP
   TRANSITION Trans3 FROM "Stations start  - wait for finish" TO "Wait for carousel - ReadyToCW"   // T3
      := "sq_carousel_insertion_st1".Done.X AND "sq_carousel_unloading_st2".Done.X AND NOT "ModeSelection_DB".mode.autoStatus.stopping AND ("AutoPositions".St1_Table1.PartPresent OR "AutoPositions".St2_Table2.PartPresent OR NOT "ModeSelection_DB".mode.autoStatus.emptying) AND "safety_signals"."5L+";
   END_TRANSITION
   STEP "Start turning - wait for carousel out of position":   // S4, max time T#10S, warning time T#7S
      supervision V := #"Start turning - wait for carousel out of position".T > #"Start turning - wait for carousel out of position".T_MAX;
          S1  S    "DevicesData".TurnTable.Commands.AutomaticMode.StartCW
          S0  R    "DevicesData".TurnTable.Commands.AutomaticMode.StartCW
   END_STEP
   TRANSITION Trans4 FROM "Start turning - wait for carousel out of position" TO "Turning - wait for carousel in position"   // T4
      := "DevicesData".TurnTable.Status.CycleRunning AND NOT "DevicesData".TurnTable.Status.CycleFinished AND NOT "DevicesData".TurnTable."I/O".Inputs.IndexerInPosition;
   END_TRANSITION
   TRANSITION Trans12 FROM "Start turning - wait for carousel out of position" TO "Turning interrupted - RESET light curtain"   // T12
      := NOT "safety_signals"."5L+";
   END_TRANSITION
   STEP "Turning - wait for carousel in position":   // S5, max time T#10S, warning time T#7S
      supervision V := #"Turning - wait for carousel in position".T > #"Turning - wait for carousel in position".T_MAX;
   END_STEP
   TRANSITION Trans5 FROM "Turning - wait for carousel in position" TO "Stations must be in base position"   // T5, jump
      := NOT "DevicesData".TurnTable.Status.CycleRunning AND "DevicesData".TurnTable.Status.CycleFinished AND "DevicesData".TurnTable."I/O".Inputs.IndexerInPosition;
   END_TRANSITION
   TRANSITION Trans13 FROM "Turning - wait for carousel in position" TO "Turning interrupted - RESET light curtain"   // T13, jump
      := NOT "safety_signals"."5L+";
   END_TRANSITION
   STEP "Turning interrupted - RESET light curtain":   // S17, max time T#10S, warning time T#7S
   END_STEP
   TRANSITION Trans14 FROM "Turning interrupted - RESET light curtain" TO "Wait for carousel - ReadyToCW"   // T14, jump
      := (#"Turning interrupted - RESET light curtain".T > t#2000MS) AND "safety_signals"."5L+" AND NOT "DevicesData".TurnTable."I/O".Inputs.IndexerInPosition;
   END_TRANSITION
   TRANSITION Trans16 FROM "Turning interrupted - RESET light curtain" TO "Turning - wait for carousel in position"   // T16, jump
      := (#"Turning interrupted - RESET light curtain".T > t#2000MS) AND "safety_signals"."5L+" AND "DevicesData".TurnTable."I/O".Inputs.IndexerInPosition;
   END_TRANSITION
   STEP "Wait for carousel - ReadyToCW":   // S18, max time T#10S, warning time T#7S
      supervision V := #"Wait for carousel - ReadyToCW".T > #"Wait for carousel - ReadyToCW".T_MAX;
   END_STEP
   TRANSITION Trans15 FROM "Wait for carousel - ReadyToCW" TO "Wait for robot out of zone"   // T15
      := "DevicesData".TurnTable.Commands.AutomaticMode.ReadyToStartCW;
   END_TRANSITION
   STEP "Wait for stations to finish base":   // S8, max time T#10S, warning time T#7S
   END_STEP
   TRANSITION Trans10 FROM "Wait for stations to finish base" TO "Wait for carousel - ReadyToCW"   // T10
      := "sq_carousel_insertion_st1"."Base done".X AND "sq_carousel_unloading_st2"."Base done".X AND "sq_robot_"."Base done".X AND "safety_signals"."5L+";
   END_TRANSITION
   STEP "auto / base":   // S20, max time T#10S, warning time T#7S
   END_STEP
   TRANSITION Trans22 FROM "auto / base" TO "Stations start  - wait for finish"   // T22
      := (("ModeSelection_DB".mode.activeMode = "mode_3_automat") OR (("ModeSelection_DB".mode.activeMode = "mode_4_semiautomat") AND #start)) AND "DevicesData".TurnTable."I/O".Inputs.IndexerInPosition;
   END_TRANSITION
   TRANSITION Trans23 FROM "auto / base" TO "Wait for stations to finish base"   // T23
      := (("ModeSelection_DB".mode.activeMode = "mode_2_base") OR (("ModeSelection_DB".mode.activeMode = "mode_4_semiautomat") AND #start)) AND NOT "DevicesData".TurnTable."I/O".Inputs.IndexerInPosition;
   END_TRANSITION
   TRANSITION Trans24 FROM "auto / base" TO "Base done"   // T24
      := ("ModeSelection_DB".mode.activeMode = "mode_2_base") AND "DevicesData".TurnTable."I/O".Inputs.IndexerInPosition;
   END_TRANSITION
   STEP "Base done":   // S14, max time T#10S, warning time T#7S
   END_STEP
   TRANSITION Trans18 FROM "Base done" TO "auto / base"   // T18, jump
      := "ModeSelection_DB".mode.activeMode = "mode_3_automat";
   END_TRANSITION
   STEP "Wait for robot out of zone":   // S15, max time T#10S, warning time T#7S
      supervision V := #"Wait for robot out of zone".T > #"Wait for robot out of zone".T_MAX;
   END_STEP
   TRANSITION Trans19 FROM "Wait for robot out of zone" TO "Start turning - wait for carousel out of position"   // T19
      := "iR1OutOfSt2";
   END_TRANSITION
END_FUNCTION_BLOCK

